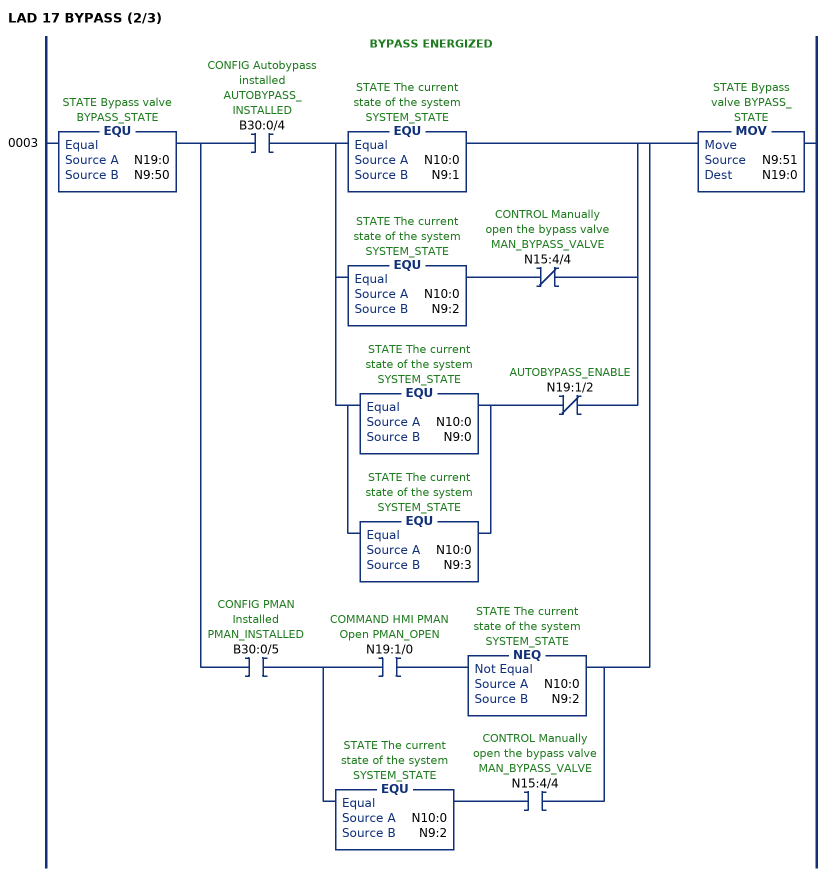
% Rung: 3 %
% TITLE: BYPASS ENERGIZED %
SOR EQU N19:0 N9:50 BST XIC B30:0/4 BST EQU N10:0 N9:1 NXB EQU N10:0 N9:2 XIO N15:4/4 NXB BST EQU N10:0 N9:0 NXB EQU N10:0 N9:3 BND XIO N19:1/2 BND NXB XIC B30:0/5 BST XIC N19:1/0 NEQ N10:0 N9:2 NXB EQU N10:0 N9:2 XIC N15:4/4 BND BND MOV N9:51 N19:0 EOR
%   N19:0  BYPASS_STATE  "STATE Bypass valve" %
%   N9:50  BYPASS_DEENERGIZED  "STATE Bypass Deenergized" %
%   B30:0/4  AUTOBYPASS_INSTALLED  "CONFIG Autobypass installed" %
%   N10:0  SYSTEM_STATE  "STATE The current state of the system" %
%   N9:1  SYSTEM_PROCESS  "STATE System Process" %
%   N9:2  SYSTEM_MANUAL  "STATE System Manual" %
%   N15:4/4  MAN_BYPASS_VALVE  "CONTROL Manually open the bypass valve" %
%   N9:0  SYSTEM_STANDBY  "STATE System Standby" %
%   N9:3  SYSTEM_ALARM  "STATE System Alarm" %
%   N19:1/2  AUTOBYPASS_ENABLE %
%   B30:0/5  PMAN_INSTALLED  "CONFIG PMAN Installed" %
%   N19:1/0  PMAN_OPEN  "COMMAND HMI PMAN Open" %
%   N9:51  BYPASS_ENERGIZED  "STATE Bypass Energized" %

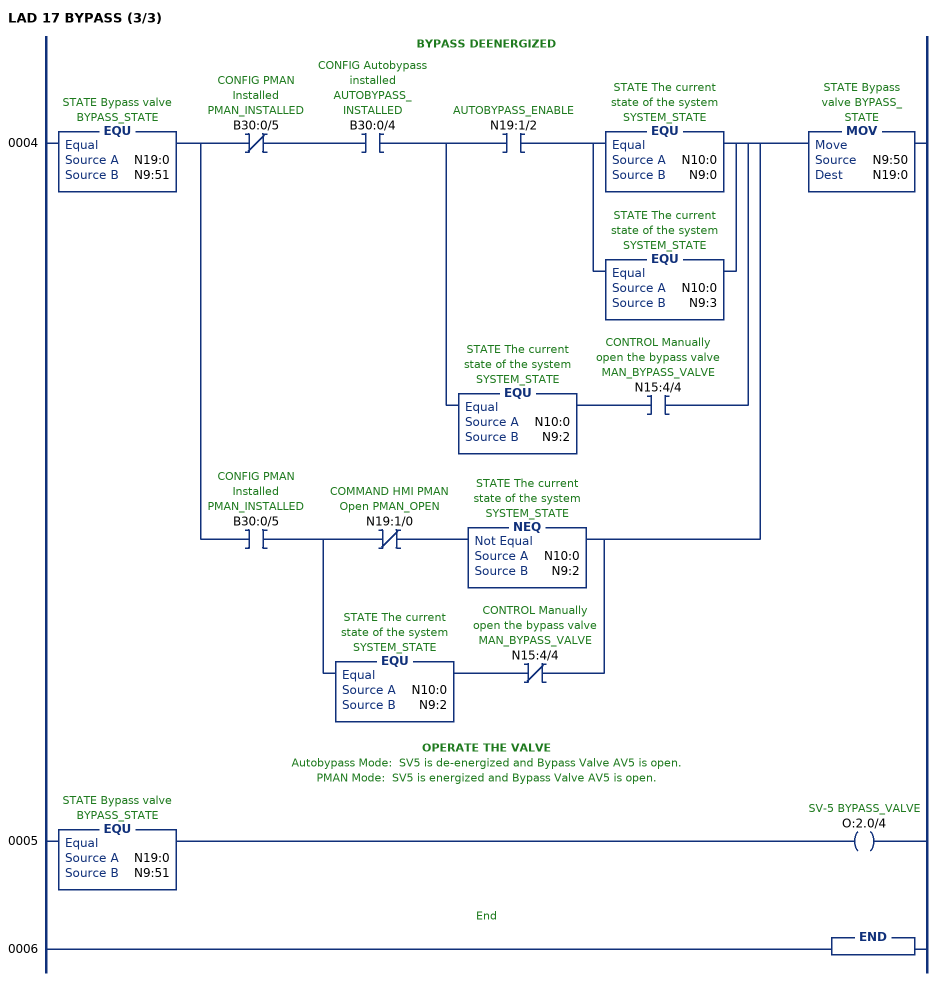
% Rung: 4 %
% TITLE: BYPASS DEENERGIZED %
SOR EQU N19:0 N9:51 BST XIO B30:0/5 XIC B30:0/4 BST XIC N19:1/2 BST EQU N10:0 N9:0 NXB EQU N10:0 N9:3 BND NXB EQU N10:0 N9:2 XIC N15:4/4 BND NXB XIC B30:0/5 BST XIO N19:1/0 NEQ N10:0 N9:2 NXB EQU N10:0 N9:2 XIO N15:4/4 BND BND MOV N9:50 N19:0 EOR
%   N19:0  BYPASS_STATE  "STATE Bypass valve" %
%   N9:51  BYPASS_ENERGIZED  "STATE Bypass Energized" %
%   B30:0/5  PMAN_INSTALLED  "CONFIG PMAN Installed" %
%   B30:0/4  AUTOBYPASS_INSTALLED  "CONFIG Autobypass installed" %
%   N19:1/2  AUTOBYPASS_ENABLE %
%   N10:0  SYSTEM_STATE  "STATE The current state of the system" %
%   N9:0  SYSTEM_STANDBY  "STATE System Standby" %
%   N9:3  SYSTEM_ALARM  "STATE System Alarm" %
%   N9:2  SYSTEM_MANUAL  "STATE System Manual" %
%   N15:4/4  MAN_BYPASS_VALVE  "CONTROL Manually open the bypass valve" %
%   N19:1/0  PMAN_OPEN  "COMMAND HMI PMAN Open" %
%   N9:50  BYPASS_DEENERGIZED  "STATE Bypass Deenergized" %
% Rung: 5 %
% TITLE: OPERATE THE VALVE %
% Autobypass Mode:  SV5 is de-energized and Bypass Valve AV5 is open.
% PMAN Mode:  SV5 is energized and Bypass Valve AV5 is open. %
SOR EQU N19:0 N9:51 OTE O:2.0/4 EOR
%   N19:0  BYPASS_STATE  "STATE Bypass valve" %
%   N9:51  BYPASS_ENERGIZED  "STATE Bypass Energized" %
%   O:2.0/4  BYPASS_VALVE  "SV-5" %
% Rung: 6 %
% End %
SOR END EOR

LADDER 18 "MIX PANEL"
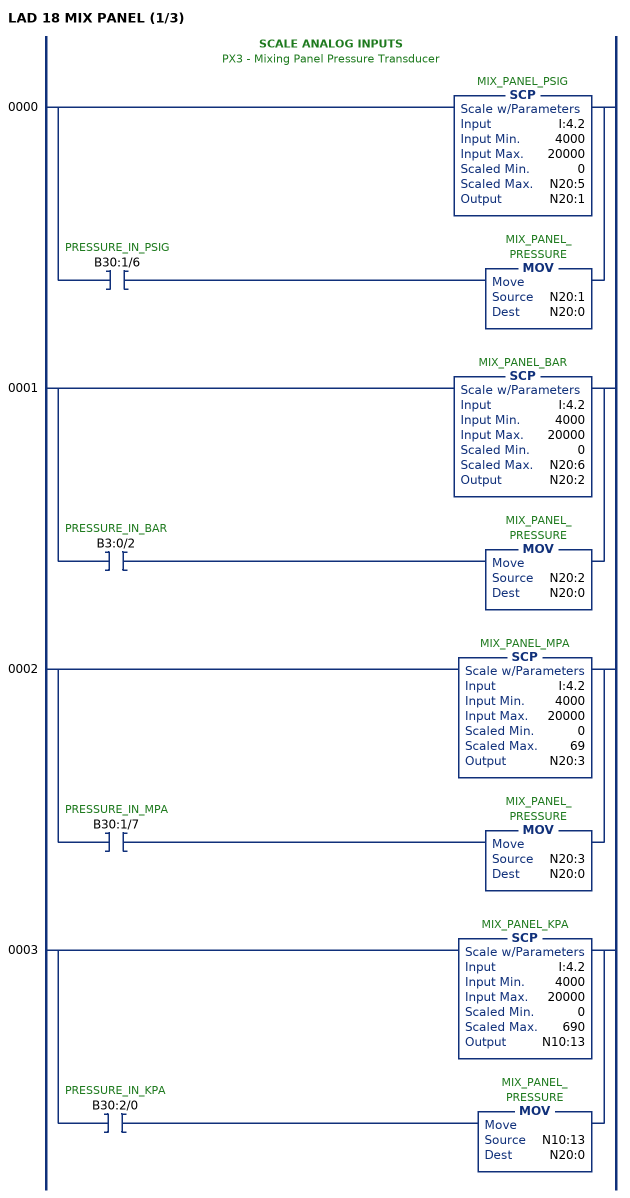
% Rung: 0 %
% TITLE: SCALE ANALOG INPUTS %
% PX3 - Mixing Panel Pressure Transducer %
SOR BST SCP I:4.2 4000 20000 0 N20:5 N20:1 NXB XIC B30:1/6 MOV N20:1 N20:0 BND EOR
%   I:4.2  MIX_PANEL_PX_READING  "PX-3" %
%   N20:5  PX3_SCALING %
%   N20:1  MIX_PANEL_PSIG %
%   B30:1/6  PRESSURE_IN_PSIG %
%   N20:0  MIX_PANEL_PRESSURE %
% Rung: 1 %
SOR BST SCP I:4.2 4000 20000 0 N20:6 N20:2 NXB XIC B3:0/2 MOV N20:2 N20:0 BND EOR
%   I:4.2  MIX_PANEL_PX_READING  "PX-3" %
%   N20:6  PX3_SCALING_BAR %
%   N20:2  MIX_PANEL_BAR %
%   B3:0/2  PRESSURE_IN_BAR %
%   N20:0  MIX_PANEL_PRESSURE %
% Rung: 2 %
SOR BST SCP I:4.2 4000 20000 0 69 N20:3 NXB XIC B30:1/7 MOV N20:3 N20:0 BND EOR
%   I:4.2  MIX_PANEL_PX_READING  "PX-3" %
%   N20:3  MIX_PANEL_MPA %
%   B30:1/7  PRESSURE_IN_MPA %
%   N20:0  MIX_PANEL_PRESSURE %
% Rung: 3 %
SOR BST SCP I:4.2 4000 20000 0 690 N10:13 NXB XIC B30:2/0 MOV N10:13 N20:0 BND EOR
%   I:4.2  MIX_PANEL_PX_READING  "PX-3" %
%   N10:13  MIX_PANEL_KPA %
%   B30:2/0  PRESSURE_IN_KPA %
%   N20:0  MIX_PANEL_PRESSURE %

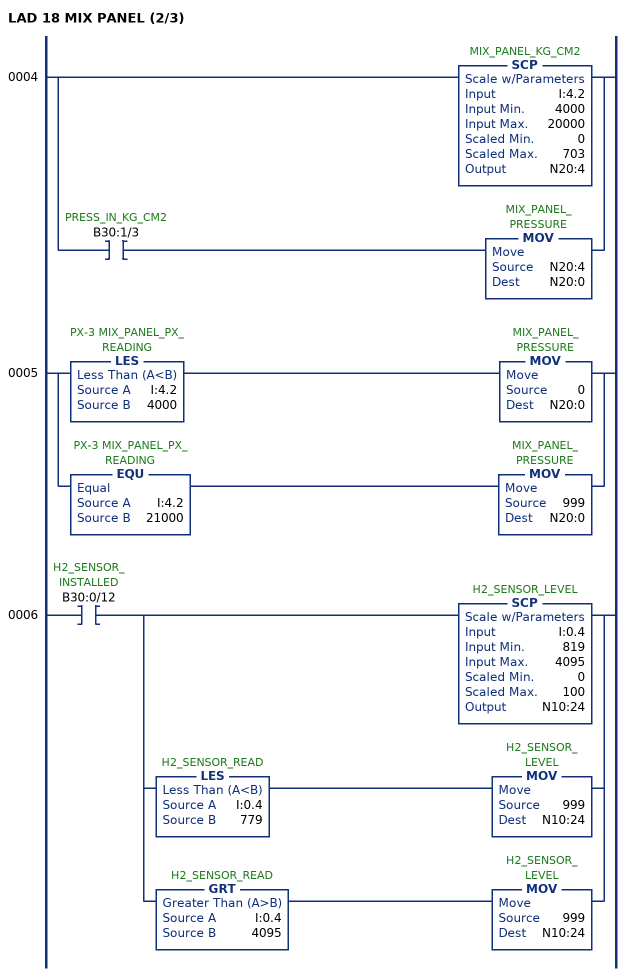
% Rung: 4 %
SOR BST SCP I:4.2 4000 20000 0 703 N20:4 NXB XIC B30:1/3 MOV N20:4 N20:0 BND EOR
%   I:4.2  MIX_PANEL_PX_READING  "PX-3" %
%   N20:4  MIX_PANEL_KG_CM2 %
%   B30:1/3  PRESS_IN_KG_CM2 %
%   N20:0  MIX_PANEL_PRESSURE %
% Rung: 5 %
SOR BST LES I:4.2 4000 MOV 0 N20:0 NXB EQU I:4.2 21000 MOV 999 N20:0 BND EOR
%   I:4.2  MIX_PANEL_PX_READING  "PX-3" %
%   N20:0  MIX_PANEL_PRESSURE %
% Rung: 6 %
SOR XIC B30:0/12 BST SCP I:0.4 819 4095 0 100 N10:24 NXB LES I:0.4 779 MOV 999 N10:24 NXB GRT I:0.4 4095 MOV 999 N10:24 BND EOR
%   B30:0/12  H2_SENSOR_INSTALLED %
%   I:0.4  H2_SENSOR_READ %
%   N10:24  H2_SENSOR_LEVEL %

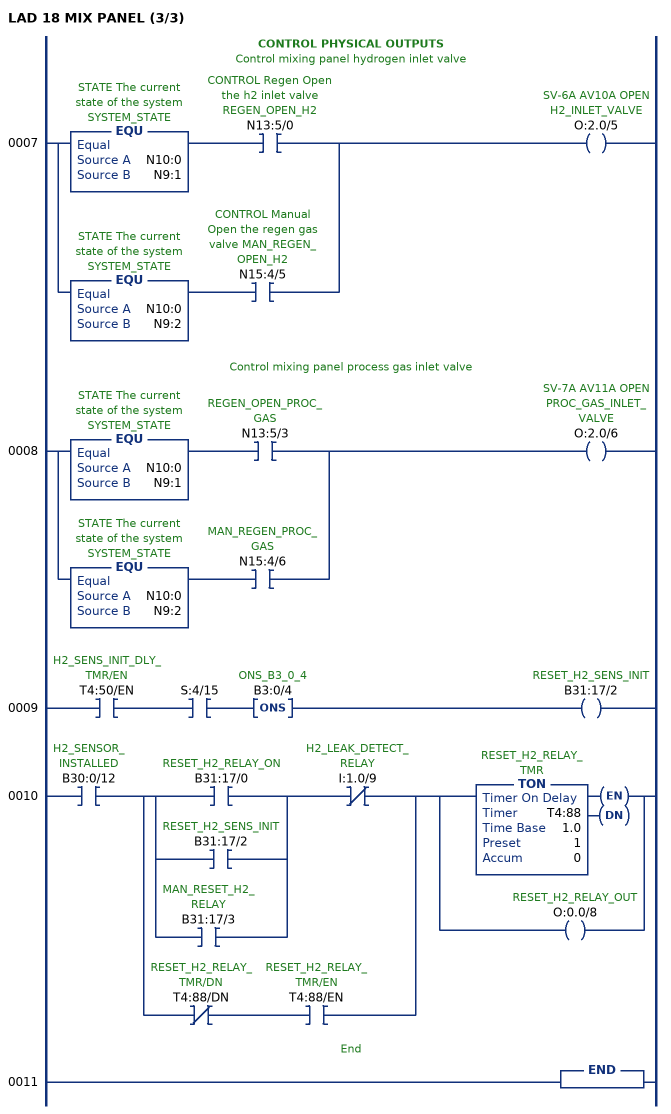
% Rung: 7 %
% TITLE: CONTROL PHYSICAL OUTPUTS %
% Control mixing panel hydrogen inlet valve %
SOR BST EQU N10:0 N9:1 XIC N13:5/0 NXB EQU N10:0 N9:2 XIC N15:4/5 BND OTE O:2.0/5 EOR
%   N10:0  SYSTEM_STATE  "STATE The current state of the system" %
%   N9:1  SYSTEM_PROCESS  "STATE System Process" %
%   N13:5/0  REGEN_OPEN_H2  "CONTROL Regen Open the h2 inlet valve" %
%   N9:2  SYSTEM_MANUAL  "STATE System Manual" %
%   N15:4/5  MAN_REGEN_OPEN_H2  "CONTROL Manual Open the regen gas valve" %
%   O:2.0/5  H2_INLET_VALVE  "SV-6A AV10A OPEN" %
% Rung: 8 %
% Control mixing panel process gas inlet valve %
SOR BST EQU N10:0 N9:1 XIC N13:5/3 NXB EQU N10:0 N9:2 XIC N15:4/6 BND OTE O:2.0/6 EOR
%   N10:0  SYSTEM_STATE  "STATE The current state of the system" %
%   N9:1  SYSTEM_PROCESS  "STATE System Process" %
%   N13:5/3  REGEN_OPEN_PROC_GAS %
%   N9:2  SYSTEM_MANUAL  "STATE System Manual" %
%   N15:4/6  MAN_REGEN_PROC_GAS %
%   O:2.0/6  PROC_GAS_INLET_VALVE  "SV-7A AV11A OPEN" %
% Rung: 9 %
SOR XIC T4:50/EN XIC S:4/15 ONS B3:0/4 OTE B31:17/2 EOR
%   T4:50  H2_SENS_INIT_DLY_TMR %
%   B3:0/4  ONS_B3_0_4 %
%   B31:17/2  RESET_H2_SENS_INIT %
% Rung: 10 %
SOR XIC B30:0/12 BST BST XIC B31:17/0 NXB XIC B31:17/2 NXB XIC B31:17/3 BND XIO I:1.0/9 NXB XIO T4:88/DN XIC T4:88/EN BND BST TON T4:88 1.0 1 0 NXB OTE O:0.0/8 BND EOR
%   B30:0/12  H2_SENSOR_INSTALLED %
%   B31:17/0  RESET_H2_RELAY_ON %
%   B31:17/2  RESET_H2_SENS_INIT %
%   B31:17/3  MAN_RESET_H2_RELAY %
%   I:1.0/9  H2_LEAK_DETECT_RELAY %
%   T4:88  RESET_H2_RELAY_TMR %
%   O:0.0/8  RESET_H2_RELAY_OUT %
% Rung: 11 %
% End %
SOR END EOR

LADDER 20 "ADS_A"    % Controls the Adsorber A %
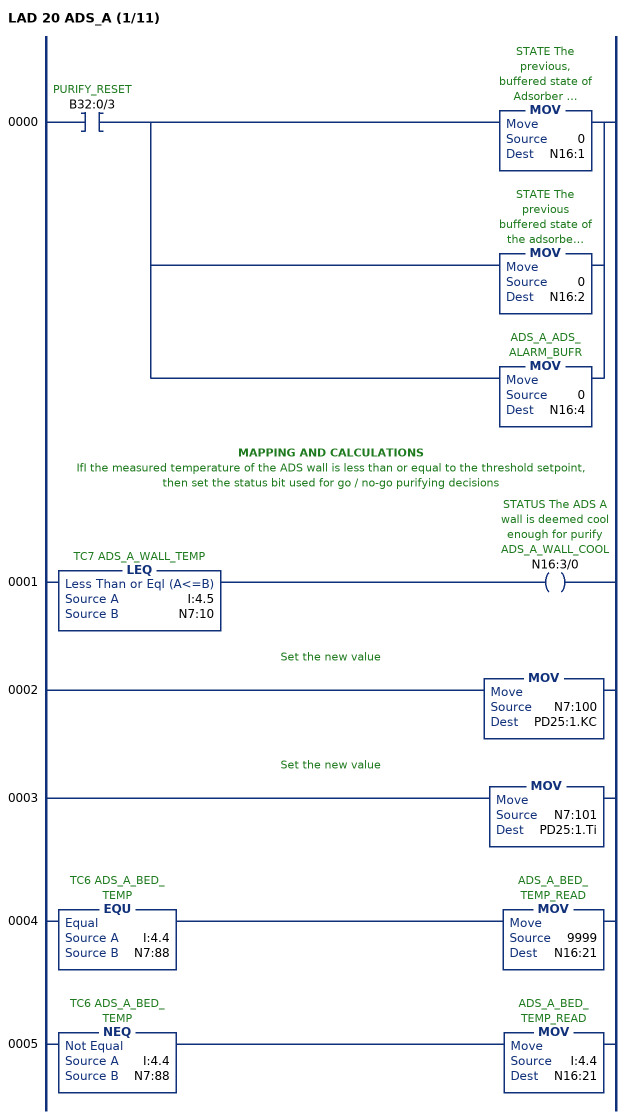
% Rung: 0 %
SOR XIC B32:0/3 BST MOV 0 N16:1 NXB MOV 0 N16:2 NXB MOV 0 N16:4 BND EOR
%   B32:0/3  PURIFY_RESET %
%   N16:1  ADS_A_STANDBY_BUFFER  "STATE The previous, buffered state of Adsorber A" %
%   N16:2  ADS_A_SYS_ALARM_BUFR  "STATE The previous buffered state of the adsorber when the alarm occured" %
%   N16:4  ADS_A_ADS_ALARM_BUFR %
% Rung: 1 %
% TITLE: MAPPING AND CALCULATIONS %
% IfI the measured temperature of the ADS wall is less than or equal to the threshold setpoint, then set the status bit used for go / no-go purifying decisions %
SOR LEQ I:4.5 N7:10 OTE N16:3/0 EOR
%   I:4.5  ADS_A_WALL_TEMP  "TC7" %
%   N7:10  ADS_WALL_TEMP_COOL  "CONFIG The temp at which the adsorber wall is deemed to be cool enough to purify" %
%   N16:3/0  ADS_A_WALL_COOL  "STATUS The ADS A wall is deemed cool enough for purify" %
% Rung: 2 %
% Set the new value %
SOR MOV N7:100 PD25:1.KC EOR
%   N7:100  BLANKET_P  "CONFIG Blanket Proportional Gain New" %
% Rung: 3 %
% Set the new value %
SOR MOV N7:101 PD25:1.Ti EOR
%   N7:101  BLANKET_I  "CONFIG Blanket Integral Gain New" %
% Rung: 4 %
SOR EQU I:4.4 N7:88 MOV 9999 N16:21 EOR
%   I:4.4  ADS_A_BED_TEMP  "TC6" %
%   N7:88  TC_OPEN_SP  "CONFIG The value read by an open TC input" %
%   N16:21  ADS_A_BED_TEMP_READ %
% Rung: 5 %
SOR NEQ I:4.4 N7:88 MOV I:4.4 N16:21 EOR
%   I:4.4  ADS_A_BED_TEMP  "TC6" %
%   N7:88  TC_OPEN_SP  "CONFIG The value read by an open TC input" %
%   N16:21  ADS_A_BED_TEMP_READ %

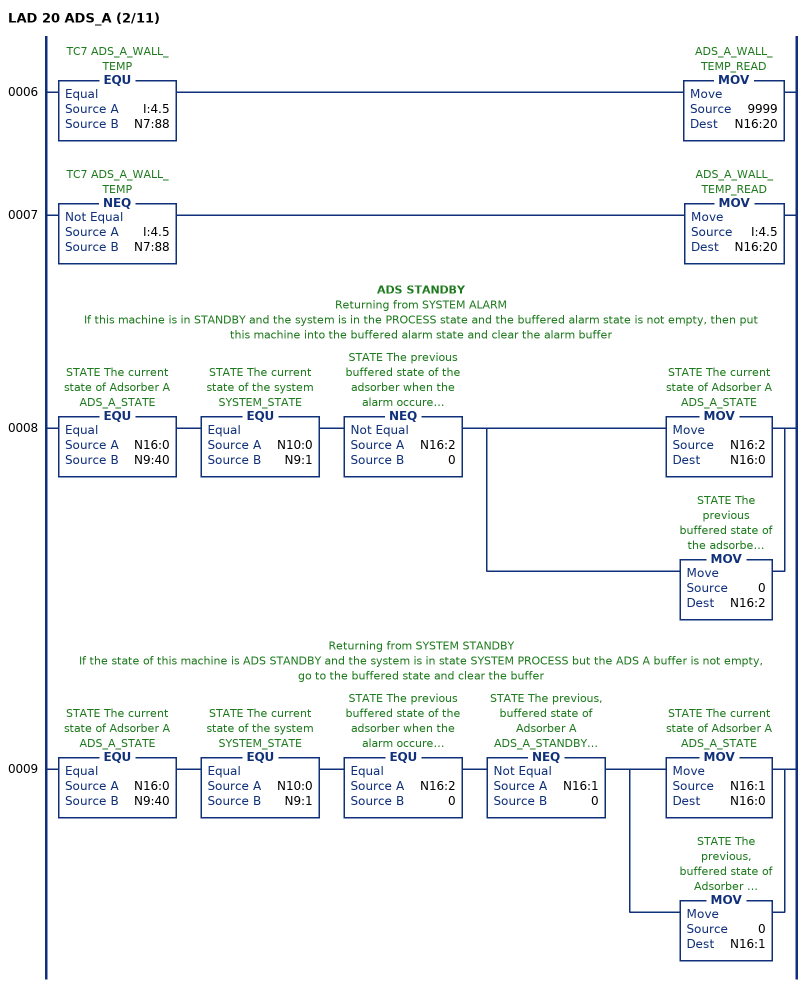
% Rung: 6 %
SOR EQU I:4.5 N7:88 MOV 9999 N16:20 EOR
%   I:4.5  ADS_A_WALL_TEMP  "TC7" %
%   N7:88  TC_OPEN_SP  "CONFIG The value read by an open TC input" %
%   N16:20  ADS_A_WALL_TEMP_READ %
% Rung: 7 %
SOR NEQ I:4.5 N7:88 MOV I:4.5 N16:20 EOR
%   I:4.5  ADS_A_WALL_TEMP  "TC7" %
%   N7:88  TC_OPEN_SP  "CONFIG The value read by an open TC input" %
%   N16:20  ADS_A_WALL_TEMP_READ %
% Rung: 8 %
% TITLE: ADS STANDBY %
% Returning from SYSTEM ALARM
% If this machine is in STANDBY and the system is in the PROCESS state and the buffered alarm state is not empty, then put this machine into the buffered alarm state and clear the alarm buffer %
SOR EQU N16:0 N9:40 EQU N10:0 N9:1 NEQ N16:2 0 BST MOV N16:2 N16:0 NXB MOV 0 N16:2 BND EOR
%   N16:0  ADS_A_STATE  "STATE The current state of Adsorber A" %
%   N9:40  ADS_STANDBY  "STATE ADS Standby" %
%   N10:0  SYSTEM_STATE  "STATE The current state of the system" %
%   N9:1  SYSTEM_PROCESS  "STATE System Process" %
%   N16:2  ADS_A_SYS_ALARM_BUFR  "STATE The previous buffered state of the adsorber when the alarm occured" %
% Rung: 9 %
% Returning from SYSTEM STANDBY
% If the state of this machine is ADS STANDBY and the system is in state SYSTEM PROCESS but the ADS A buffer is not empty, go to the buffered state and clear the buffer %
SOR EQU N16:0 N9:40 EQU N10:0 N9:1 EQU N16:2 0 NEQ N16:1 0 BST MOV N16:1 N16:0 NXB MOV 0 N16:1 BND EOR
%   N16:0  ADS_A_STATE  "STATE The current state of Adsorber A" %
%   N9:40  ADS_STANDBY  "STATE ADS Standby" %
%   N10:0  SYSTEM_STATE  "STATE The current state of the system" %
%   N9:1  SYSTEM_PROCESS  "STATE System Process" %
%   N16:2  ADS_A_SYS_ALARM_BUFR  "STATE The previous buffered state of the adsorber when the alarm occured" %
%   N16:1  ADS_A_STANDBY_BUFFER  "STATE The previous, buffered state of Adsorber A" %

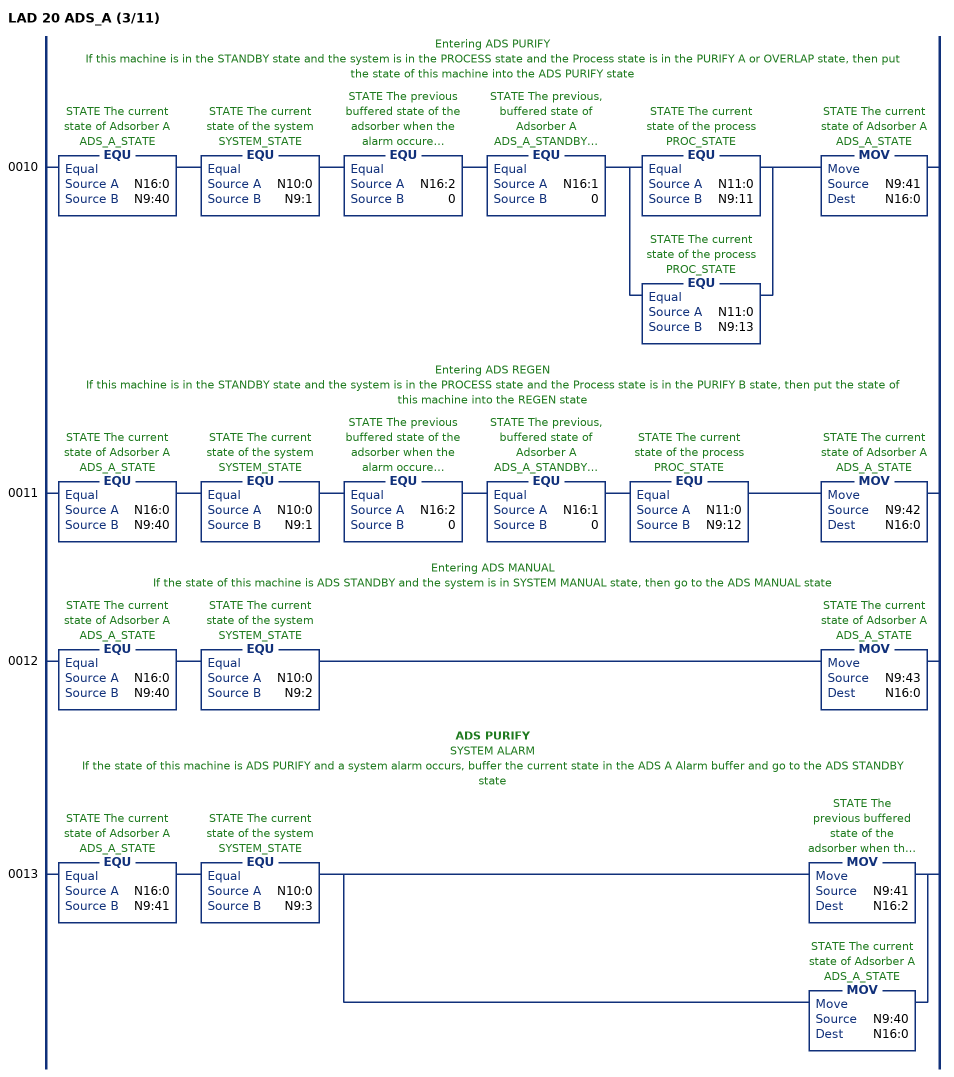
% Rung: 10 %
% Entering ADS PURIFY
% If this machine is in the STANDBY state and the system is in the PROCESS state and the Process state is in the PURIFY A or OVERLAP state, then put the state of this machine into the ADS PURIFY state %
SOR EQU N16:0 N9:40 EQU N10:0 N9:1 EQU N16:2 0 EQU N16:1 0 BST EQU N11:0 N9:11 NXB EQU N11:0 N9:13 BND MOV N9:41 N16:0 EOR
%   N16:0  ADS_A_STATE  "STATE The current state of Adsorber A" %
%   N9:40  ADS_STANDBY  "STATE ADS Standby" %
%   N10:0  SYSTEM_STATE  "STATE The current state of the system" %
%   N9:1  SYSTEM_PROCESS  "STATE System Process" %
%   N16:2  ADS_A_SYS_ALARM_BUFR  "STATE The previous buffered state of the adsorber when the alarm occured" %
%   N16:1  ADS_A_STANDBY_BUFFER  "STATE The previous, buffered state of Adsorber A" %
%   N11:0  PROC_STATE  "STATE The current state of the process" %
%   N9:11  PROC_PURIFY_A  "STATE Process Purify A" %
%   N9:13  PROC_OVERLAP  "STATE Process Purify Overlap" %
%   N9:41  ADS_PURIFY  "STATE ADS Purify" %
% Rung: 11 %
% Entering ADS REGEN
% If this machine is in the STANDBY state and the system is in the PROCESS state and the Process state is in the PURIFY B state, then put the state of this machine into the REGEN state %
SOR EQU N16:0 N9:40 EQU N10:0 N9:1 EQU N16:2 0 EQU N16:1 0 EQU N11:0 N9:12 MOV N9:42 N16:0 EOR
%   N16:0  ADS_A_STATE  "STATE The current state of Adsorber A" %
%   N9:40  ADS_STANDBY  "STATE ADS Standby" %
%   N10:0  SYSTEM_STATE  "STATE The current state of the system" %
%   N9:1  SYSTEM_PROCESS  "STATE System Process" %
%   N16:2  ADS_A_SYS_ALARM_BUFR  "STATE The previous buffered state of the adsorber when the alarm occured" %
%   N16:1  ADS_A_STANDBY_BUFFER  "STATE The previous, buffered state of Adsorber A" %
%   N11:0  PROC_STATE  "STATE The current state of the process" %
%   N9:12  PROC_PURIFY_B  "STATE Process Purify B" %
%   N9:42  ADS_REGEN  "STATE ADS Regen" %
% Rung: 12 %
% Entering ADS MANUAL
% If the state of this machine is ADS STANDBY and the system is in SYSTEM MANUAL state, then go to the ADS MANUAL state %
SOR EQU N16:0 N9:40 EQU N10:0 N9:2 MOV N9:43 N16:0 EOR
%   N16:0  ADS_A_STATE  "STATE The current state of Adsorber A" %
%   N9:40  ADS_STANDBY  "STATE ADS Standby" %
%   N10:0  SYSTEM_STATE  "STATE The current state of the system" %
%   N9:2  SYSTEM_MANUAL  "STATE System Manual" %
%   N9:43  ADS_MANUAL  "STATE ADS Manual" %
% Rung: 13 %
% TITLE: ADS PURIFY %
% SYSTEM ALARM
% If the state of this machine is ADS PURIFY and a system alarm occurs, buffer the current state in the ADS A Alarm buffer and go to the ADS STANDBY state %
SOR EQU N16:0 N9:41 EQU N10:0 N9:3 BST MOV N9:41 N16:2 NXB MOV N9:40 N16:0 BND EOR
%   N16:0  ADS_A_STATE  "STATE The current state of Adsorber A" %
%   N9:41  ADS_PURIFY  "STATE ADS Purify" %
%   N10:0  SYSTEM_STATE  "STATE The current state of the system" %
%   N9:3  SYSTEM_ALARM  "STATE System Alarm" %
%   N16:2  ADS_A_SYS_ALARM_BUFR  "STATE The previous buffered state of the adsorber when the alarm occured" %
%   N9:40  ADS_STANDBY  "STATE ADS Standby" %

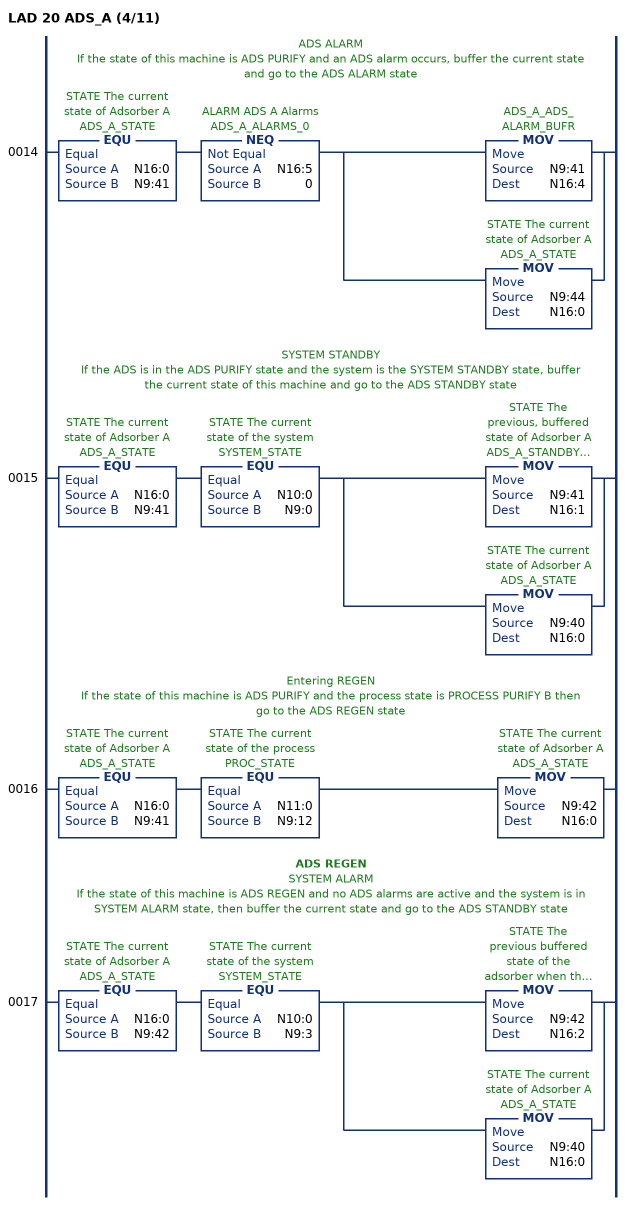
% Rung: 14 %
% ADS ALARM
% If the state of this machine is ADS PURIFY and an ADS alarm occurs, buffer the current state and go to the ADS ALARM state %
SOR EQU N16:0 N9:41 NEQ N16:5 0 BST MOV N9:41 N16:4 NXB MOV N9:44 N16:0 BND EOR
%   N16:0  ADS_A_STATE  "STATE The current state of Adsorber A" %
%   N9:41  ADS_PURIFY  "STATE ADS Purify" %
%   N16:5  ADS_A_ALARMS_0  "ALARM ADS A Alarms" %
%   N16:4  ADS_A_ADS_ALARM_BUFR %
%   N9:44  ADS_ALARM  "STATE ADS Alarm" %
% Rung: 15 %
% SYSTEM STANDBY
% If the ADS is in the ADS PURIFY state and the system is the SYSTEM STANDBY state, buffer the current state of this machine and go to the ADS STANDBY state %
SOR EQU N16:0 N9:41 EQU N10:0 N9:0 BST MOV N9:41 N16:1 NXB MOV N9:40 N16:0 BND EOR
%   N16:0  ADS_A_STATE  "STATE The current state of Adsorber A" %
%   N9:41  ADS_PURIFY  "STATE ADS Purify" %
%   N10:0  SYSTEM_STATE  "STATE The current state of the system" %
%   N9:0  SYSTEM_STANDBY  "STATE System Standby" %
%   N16:1  ADS_A_STANDBY_BUFFER  "STATE The previous, buffered state of Adsorber A" %
%   N9:40  ADS_STANDBY  "STATE ADS Standby" %
% Rung: 16 %
% Entering REGEN
% If the state of this machine is ADS PURIFY and the process state is PROCESS PURIFY B then go to the ADS REGEN state %
SOR EQU N16:0 N9:41 EQU N11:0 N9:12 MOV N9:42 N16:0 EOR
%   N16:0  ADS_A_STATE  "STATE The current state of Adsorber A" %
%   N9:41  ADS_PURIFY  "STATE ADS Purify" %
%   N11:0  PROC_STATE  "STATE The current state of the process" %
%   N9:12  PROC_PURIFY_B  "STATE Process Purify B" %
%   N9:42  ADS_REGEN  "STATE ADS Regen" %
% Rung: 17 %
% TITLE: ADS REGEN %
% SYSTEM ALARM
% If the state of this machine is ADS REGEN and no ADS alarms are active and the system is in SYSTEM ALARM state, then buffer the current state and go to the ADS STANDBY state %
SOR EQU N16:0 N9:42 EQU N10:0 N9:3 BST MOV N9:42 N16:2 NXB MOV N9:40 N16:0 BND EOR
%   N16:0  ADS_A_STATE  "STATE The current state of Adsorber A" %
%   N9:42  ADS_REGEN  "STATE ADS Regen" %
%   N10:0  SYSTEM_STATE  "STATE The current state of the system" %
%   N9:3  SYSTEM_ALARM  "STATE System Alarm" %
%   N16:2  ADS_A_SYS_ALARM_BUFR  "STATE The previous buffered state of the adsorber when the alarm occured" %
%   N9:40  ADS_STANDBY  "STATE ADS Standby" %

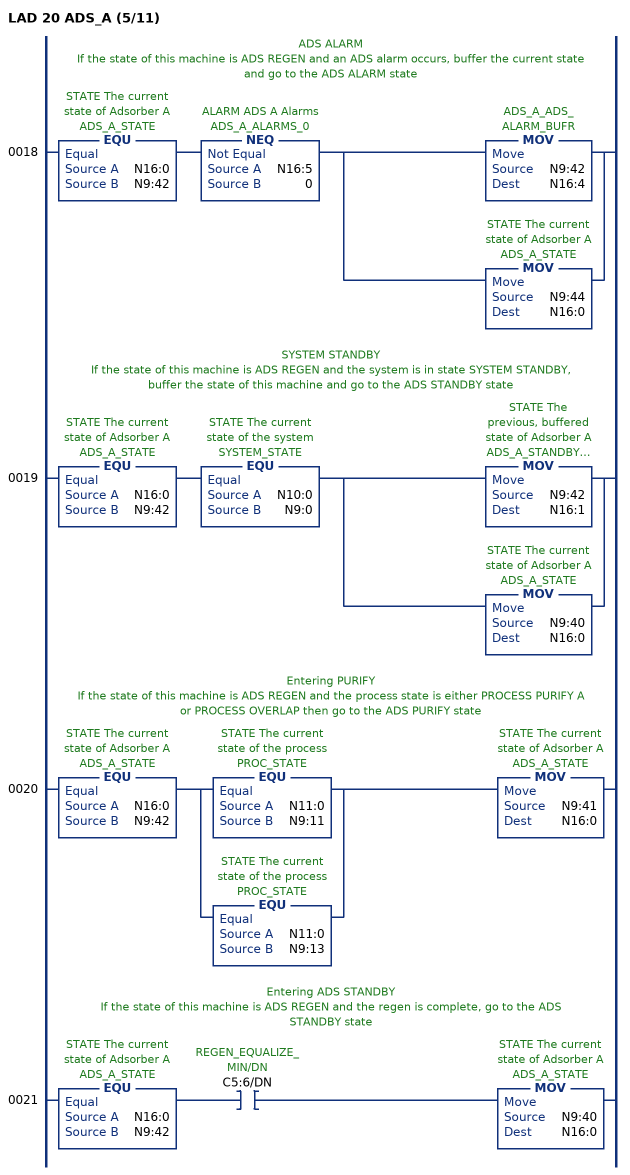
% Rung: 18 %
% ADS ALARM
% If the state of this machine is ADS REGEN and an ADS alarm occurs, buffer the current state and go to the ADS ALARM state %
SOR EQU N16:0 N9:42 NEQ N16:5 0 BST MOV N9:42 N16:4 NXB MOV N9:44 N16:0 BND EOR
%   N16:0  ADS_A_STATE  "STATE The current state of Adsorber A" %
%   N9:42  ADS_REGEN  "STATE ADS Regen" %
%   N16:5  ADS_A_ALARMS_0  "ALARM ADS A Alarms" %
%   N16:4  ADS_A_ADS_ALARM_BUFR %
%   N9:44  ADS_ALARM  "STATE ADS Alarm" %
% Rung: 19 %
% SYSTEM STANDBY
% If the state of this machine is ADS REGEN and the system is in state SYSTEM STANDBY, buffer the state of this machine and go to the ADS STANDBY state %
SOR EQU N16:0 N9:42 EQU N10:0 N9:0 BST MOV N9:42 N16:1 NXB MOV N9:40 N16:0 BND EOR
%   N16:0  ADS_A_STATE  "STATE The current state of Adsorber A" %
%   N9:42  ADS_REGEN  "STATE ADS Regen" %
%   N10:0  SYSTEM_STATE  "STATE The current state of the system" %
%   N9:0  SYSTEM_STANDBY  "STATE System Standby" %
%   N16:1  ADS_A_STANDBY_BUFFER  "STATE The previous, buffered state of Adsorber A" %
%   N9:40  ADS_STANDBY  "STATE ADS Standby" %
% Rung: 20 %
% Entering PURIFY
% If the state of this machine is ADS REGEN and the process state is either PROCESS PURIFY A or PROCESS OVERLAP then go to the ADS PURIFY state %
SOR EQU N16:0 N9:42 BST EQU N11:0 N9:11 NXB EQU N11:0 N9:13 BND MOV N9:41 N16:0 EOR
%   N16:0  ADS_A_STATE  "STATE The current state of Adsorber A" %
%   N9:42  ADS_REGEN  "STATE ADS Regen" %
%   N11:0  PROC_STATE  "STATE The current state of the process" %
%   N9:11  PROC_PURIFY_A  "STATE Process Purify A" %
%   N9:13  PROC_OVERLAP  "STATE Process Purify Overlap" %
%   N9:41  ADS_PURIFY  "STATE ADS Purify" %
% Rung: 21 %
% Entering ADS STANDBY
% If the state of this machine is ADS REGEN and the regen is complete, go to the ADS STANDBY state %
SOR EQU N16:0 N9:42 XIC C5:6/DN MOV N9:40 N16:0 EOR
%   N16:0  ADS_A_STATE  "STATE The current state of Adsorber A" %
%   N9:42  ADS_REGEN  "STATE ADS Regen" %
%   C5:6  REGEN_EQUALIZE_MIN %
%   N9:40  ADS_STANDBY  "STATE ADS Standby" %

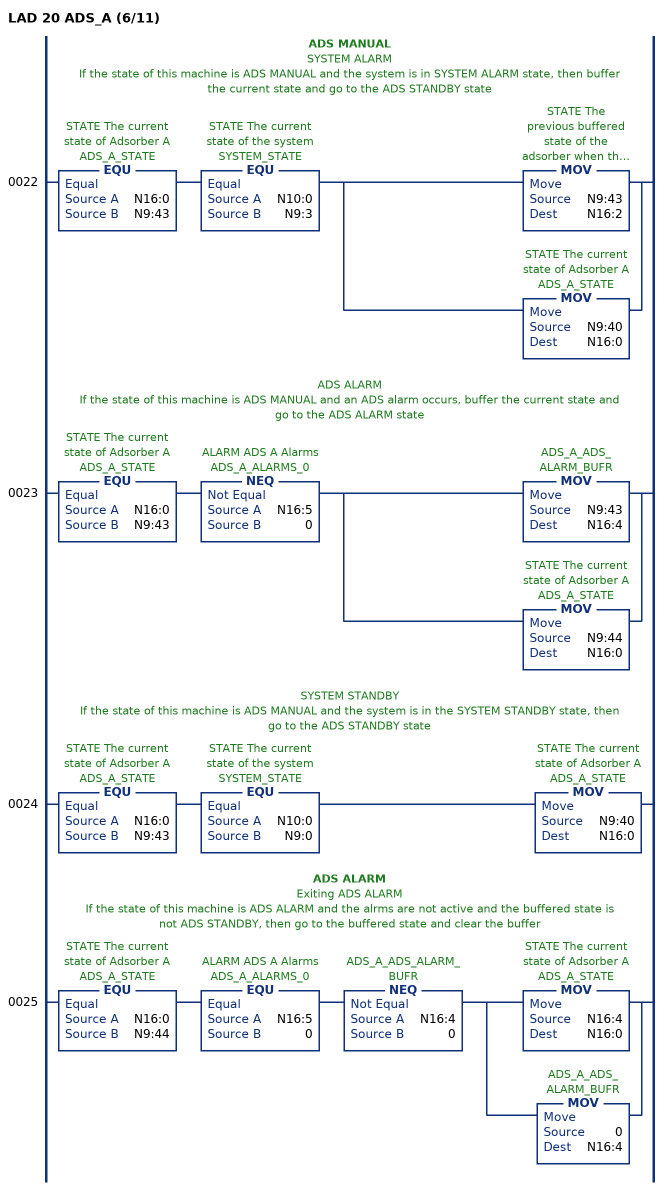
% Rung: 22 %
% TITLE: ADS MANUAL %
% SYSTEM ALARM
% If the state of this machine is ADS MANUAL and the system is in SYSTEM ALARM state, then buffer the current state and go to the ADS STANDBY state %
SOR EQU N16:0 N9:43 EQU N10:0 N9:3 BST MOV N9:43 N16:2 NXB MOV N9:40 N16:0 BND EOR
%   N16:0  ADS_A_STATE  "STATE The current state of Adsorber A" %
%   N9:43  ADS_MANUAL  "STATE ADS Manual" %
%   N10:0  SYSTEM_STATE  "STATE The current state of the system" %
%   N9:3  SYSTEM_ALARM  "STATE System Alarm" %
%   N16:2  ADS_A_SYS_ALARM_BUFR  "STATE The previous buffered state of the adsorber when the alarm occured" %
%   N9:40  ADS_STANDBY  "STATE ADS Standby" %
% Rung: 23 %
% ADS ALARM
% If the state of this machine is ADS MANUAL and an ADS alarm occurs, buffer the current state and go to the ADS ALARM state %
SOR EQU N16:0 N9:43 NEQ N16:5 0 BST MOV N9:43 N16:4 NXB MOV N9:44 N16:0 BND EOR
%   N16:0  ADS_A_STATE  "STATE The current state of Adsorber A" %
%   N9:43  ADS_MANUAL  "STATE ADS Manual" %
%   N16:5  ADS_A_ALARMS_0  "ALARM ADS A Alarms" %
%   N16:4  ADS_A_ADS_ALARM_BUFR %
%   N9:44  ADS_ALARM  "STATE ADS Alarm" %
% Rung: 24 %
% SYSTEM STANDBY
% If the state of this machine is ADS MANUAL and the system is in the SYSTEM STANDBY state, then go to the ADS STANDBY state %
SOR EQU N16:0 N9:43 EQU N10:0 N9:0 MOV N9:40 N16:0 EOR
%   N16:0  ADS_A_STATE  "STATE The current state of Adsorber A" %
%   N9:43  ADS_MANUAL  "STATE ADS Manual" %
%   N10:0  SYSTEM_STATE  "STATE The current state of the system" %
%   N9:0  SYSTEM_STANDBY  "STATE System Standby" %
%   N9:40  ADS_STANDBY  "STATE ADS Standby" %
% Rung: 25 %
% TITLE: ADS ALARM %
% Exiting ADS ALARM
% If the state of this machine is ADS ALARM and the alrms are not active and the buffered state is not ADS STANDBY, then go to the buffered state and clear the buffer %
SOR EQU N16:0 N9:44 EQU N16:5 0 NEQ N16:4 0 BST MOV N16:4 N16:0 NXB MOV 0 N16:4 BND EOR
%   N16:0  ADS_A_STATE  "STATE The current state of Adsorber A" %
%   N9:44  ADS_ALARM  "STATE ADS Alarm" %
%   N16:5  ADS_A_ALARMS_0  "ALARM ADS A Alarms" %
%   N16:4  ADS_A_ADS_ALARM_BUFR %

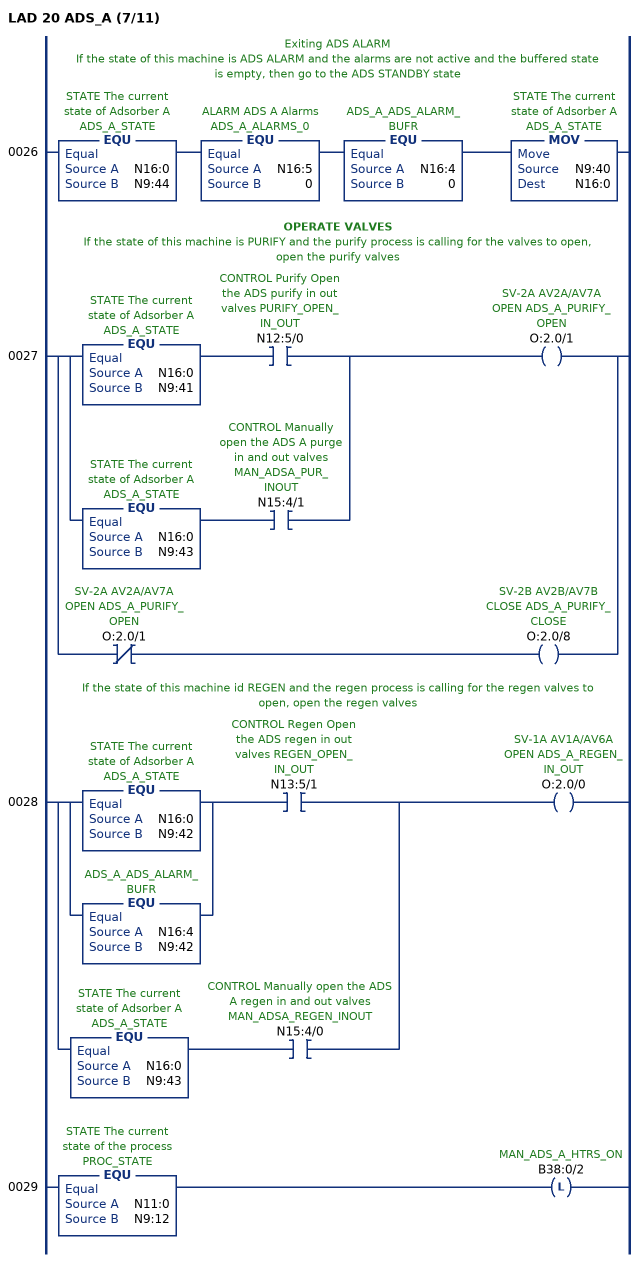
% Rung: 26 %
% Exiting ADS ALARM
% If the state of this machine is ADS ALARM and the alarms are not active and the buffered state is empty, then go to the ADS STANDBY state %
SOR EQU N16:0 N9:44 EQU N16:5 0 EQU N16:4 0 MOV N9:40 N16:0 EOR
%   N16:0  ADS_A_STATE  "STATE The current state of Adsorber A" %
%   N9:44  ADS_ALARM  "STATE ADS Alarm" %
%   N16:5  ADS_A_ALARMS_0  "ALARM ADS A Alarms" %
%   N16:4  ADS_A_ADS_ALARM_BUFR %
%   N9:40  ADS_STANDBY  "STATE ADS Standby" %
% Rung: 27 %
% TITLE: OPERATE VALVES %
% If the state of this machine is PURIFY and the purify process is calling for the valves to open, open the purify valves %
SOR BST BST EQU N16:0 N9:41 XIC N12:5/0 NXB EQU N16:0 N9:43 XIC N15:4/1 BND OTE O:2.0/1 NXB XIO O:2.0/1 OTE O:2.0/8 BND EOR
%   N16:0  ADS_A_STATE  "STATE The current state of Adsorber A" %
%   N9:41  ADS_PURIFY  "STATE ADS Purify" %
%   N12:5/0  PURIFY_OPEN_IN_OUT  "CONTROL Purify Open the ADS purify in out valves" %
%   N9:43  ADS_MANUAL  "STATE ADS Manual" %
%   N15:4/1  MAN_ADSA_PUR_INOUT  "CONTROL Manually open the ADS A purge in and out valves" %
%   O:2.0/1  ADS_A_PURIFY_OPEN  "SV-2A AV2A/AV7A OPEN" %
%   O:2.0/8  ADS_A_PURIFY_CLOSE  "SV-2B AV2B/AV7B CLOSE" %
% Rung: 28 %
% If the state of this machine id REGEN and the regen process is calling for the regen valves to open, open the regen valves %
SOR BST BST EQU N16:0 N9:42 NXB EQU N16:4 N9:42 BND XIC N13:5/1 NXB EQU N16:0 N9:43 XIC N15:4/0 BND OTE O:2.0/0 EOR
%   N16:0  ADS_A_STATE  "STATE The current state of Adsorber A" %
%   N9:42  ADS_REGEN  "STATE ADS Regen" %
%   N16:4  ADS_A_ADS_ALARM_BUFR %
%   N13:5/1  REGEN_OPEN_IN_OUT  "CONTROL Regen Open the ADS regen in out valves" %
%   N9:43  ADS_MANUAL  "STATE ADS Manual" %
%   N15:4/0  MAN_ADSA_REGEN_INOUT  "CONTROL Manually open the ADS A regen in and out valves" %
%   O:2.0/0  ADS_A_REGEN_IN_OUT  "SV-1A AV1A/AV6A OPEN" %
% Rung: 29 %
SOR EQU N11:0 N9:12 OTL B38:0/2 EOR
%   N11:0  PROC_STATE  "STATE The current state of the process" %
%   N9:12  PROC_PURIFY_B  "STATE Process Purify B" %
%   B38:0/2  MAN_ADS_A_HTRS_ON %

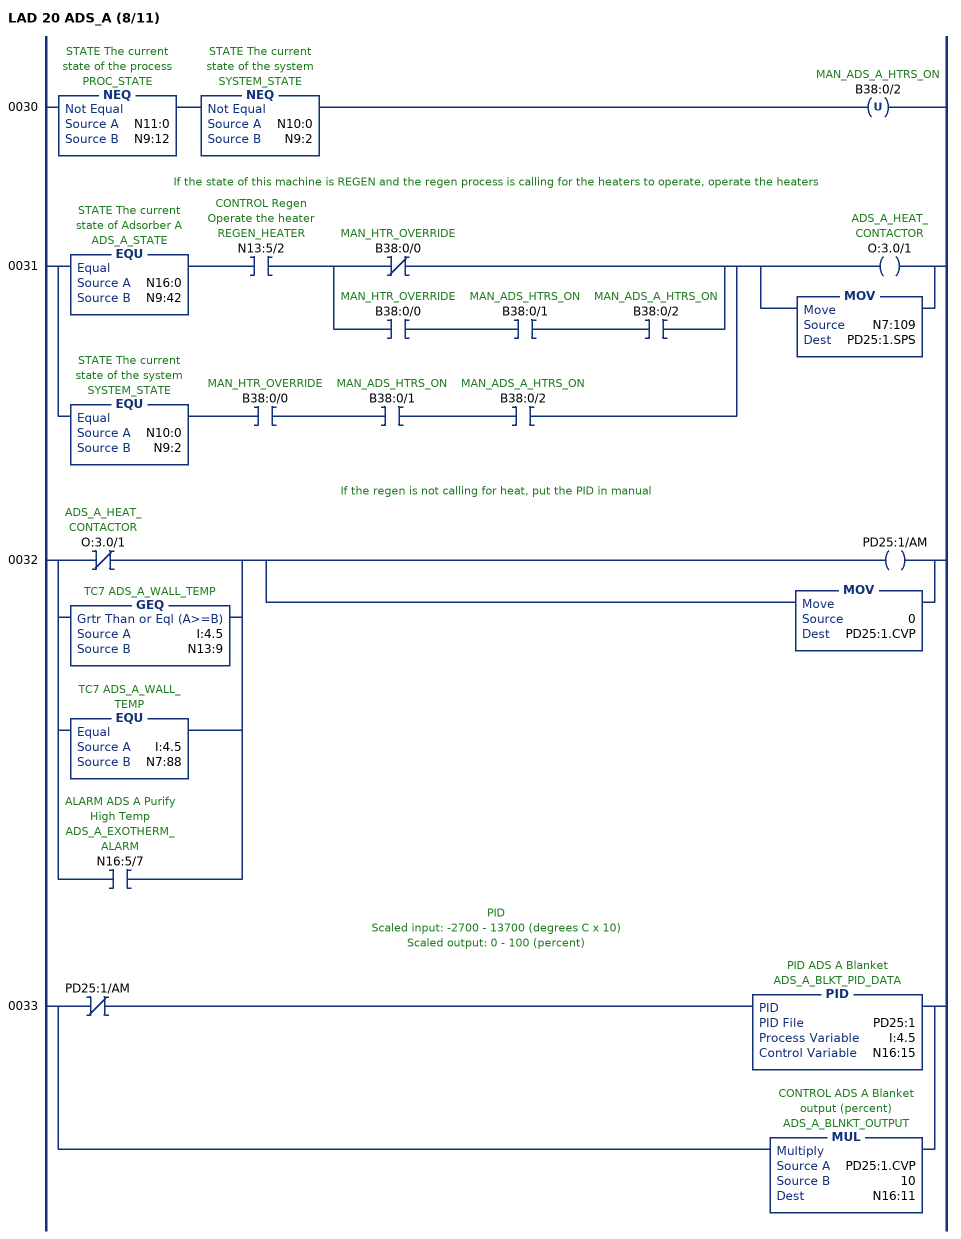
% Rung: 30 %
SOR NEQ N11:0 N9:12 NEQ N10:0 N9:2 OTU B38:0/2 EOR
%   N11:0  PROC_STATE  "STATE The current state of the process" %
%   N9:12  PROC_PURIFY_B  "STATE Process Purify B" %
%   N10:0  SYSTEM_STATE  "STATE The current state of the system" %
%   N9:2  SYSTEM_MANUAL  "STATE System Manual" %
%   B38:0/2  MAN_ADS_A_HTRS_ON %
% Rung: 31 %
% If the state of this machine is REGEN and the regen process is calling for the heaters to operate, operate the heaters %
SOR BST EQU N16:0 N9:42 XIC N13:5/2 BST XIO B38:0/0 NXB XIC B38:0/0 XIC B38:0/1 XIC B38:0/2 BND NXB EQU N10:0 N9:2 XIC B38:0/0 XIC B38:0/1 XIC B38:0/2 BND BST OTE O:3.0/1 NXB MOV N7:109 PD25:1.SPS BND EOR
%   N16:0  ADS_A_STATE  "STATE The current state of Adsorber A" %
%   N9:42  ADS_REGEN  "STATE ADS Regen" %
%   N13:5/2  REGEN_HEATER  "CONTROL Regen Operate the heater" %
%   B38:0/0  MAN_HTR_OVERRIDE %
%   B38:0/1  MAN_ADS_HTRS_ON %
%   B38:0/2  MAN_ADS_A_HTRS_ON %
%   N10:0  SYSTEM_STATE  "STATE The current state of the system" %
%   N9:2  SYSTEM_MANUAL  "STATE System Manual" %
%   O:3.0/1  ADS_A_HEAT_CONTACTOR %
%   N7:109  BLANKET_SP  "CONTROL Blanket PID Setpoint" %
% Rung: 32 %
% If the regen is not calling for heat, put the PID in manual %
SOR BST XIO O:3.0/1 NXB GEQ I:4.5 N13:9 NXB EQU I:4.5 N7:88 NXB XIC N16:5/7 BND BST OTE PD25:1/AM NXB MOV 0 PD25:1.CVP BND EOR
%   O:3.0/1  ADS_A_HEAT_CONTACTOR %
%   I:4.5  ADS_A_WALL_TEMP  "TC7" %
%   N13:9  BLANKET_LIMIT %
%   N7:88  TC_OPEN_SP  "CONFIG The value read by an open TC input" %
%   N16:5/7  ADS_A_EXOTHERM_ALARM  "ALARM ADS A Purify High Temp" %
% Rung: 33 %
% PID
% Scaled input: -2700 - 13700 (degrees C x 10)
% Scaled output: 0 - 100 (percent) %
SOR BST XIO PD25:1/AM PID PD25:1 I:4.5 N16:15 NXB MUL PD25:1.CVP 10 N16:11 BND EOR
%   PD25:1  ADS_A_BLKT_PID_DATA  "PID ADS A Blanket" %
%   I:4.5  ADS_A_WALL_TEMP  "TC7" %
%   N16:15  ADS_A_BLKT_OUTPT_RAW  "CONTROL ADS A Blanket PID Output Raw" %
%   N16:11  ADS_A_BLNKT_OUTPUT  "CONTROL ADS A Blanket output (percent)" %

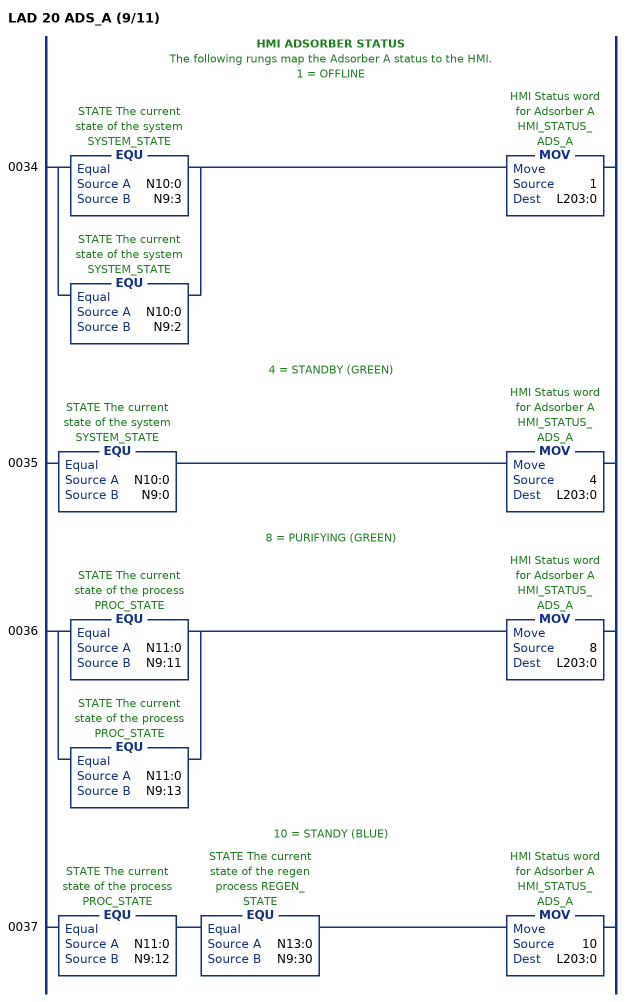
% Rung: 34 %
% TITLE: HMI ADSORBER STATUS %
% The following rungs map the Adsorber A status to the HMI.
% 1 = OFFLINE %
SOR BST EQU N10:0 N9:3 NXB EQU N10:0 N9:2 BND MOV 1 L203:0 EOR
%   N10:0  SYSTEM_STATE  "STATE The current state of the system" %
%   N9:3  SYSTEM_ALARM  "STATE System Alarm" %
%   N9:2  SYSTEM_MANUAL  "STATE System Manual" %
%   L203:0  HMI_STATUS_ADS_A  "HMI Status word for Adsorber A" %
% Rung: 35 %
% 4 = STANDBY (GREEN) %
SOR EQU N10:0 N9:0 MOV 4 L203:0 EOR
%   N10:0  SYSTEM_STATE  "STATE The current state of the system" %
%   N9:0  SYSTEM_STANDBY  "STATE System Standby" %
%   L203:0  HMI_STATUS_ADS_A  "HMI Status word for Adsorber A" %
% Rung: 36 %
% 8 = PURIFYING (GREEN) %
SOR BST EQU N11:0 N9:11 NXB EQU N11:0 N9:13 BND MOV 8 L203:0 EOR
%   N11:0  PROC_STATE  "STATE The current state of the process" %
%   N9:11  PROC_PURIFY_A  "STATE Process Purify A" %
%   N9:13  PROC_OVERLAP  "STATE Process Purify Overlap" %
%   L203:0  HMI_STATUS_ADS_A  "HMI Status word for Adsorber A" %
% Rung: 37 %
% 10 = STANDY (BLUE) %
SOR EQU N11:0 N9:12 EQU N13:0 N9:30 MOV 10 L203:0 EOR
%   N11:0  PROC_STATE  "STATE The current state of the process" %
%   N9:12  PROC_PURIFY_B  "STATE Process Purify B" %
%   N13:0  REGEN_STATE  "STATE The current state of the regen process" %
%   N9:30  REGEN_STANDBY  "STATE Regen Standby" %
%   L203:0  HMI_STATUS_ADS_A  "HMI Status word for Adsorber A" %

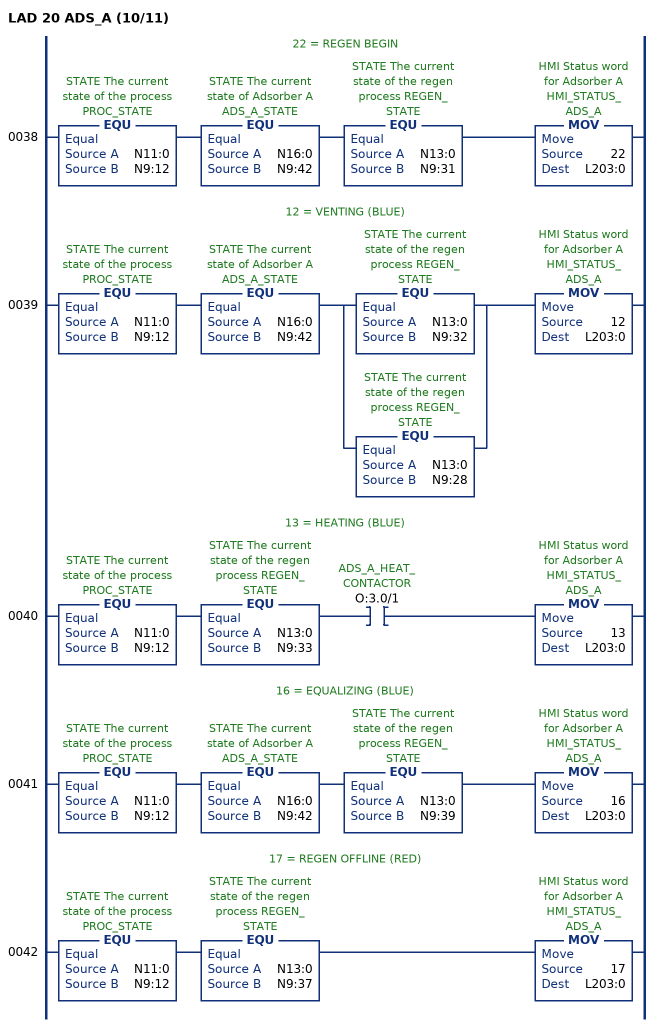
% Rung: 38 %
% 22 = REGEN BEGIN %
SOR EQU N11:0 N9:12 EQU N16:0 N9:42 EQU N13:0 N9:31 MOV 22 L203:0 EOR
%   N11:0  PROC_STATE  "STATE The current state of the process" %
%   N9:12  PROC_PURIFY_B  "STATE Process Purify B" %
%   N16:0  ADS_A_STATE  "STATE The current state of Adsorber A" %
%   N9:42  ADS_REGEN  "STATE ADS Regen" %
%   N13:0  REGEN_STATE  "STATE The current state of the regen process" %
%   N9:31  REGEN_DELAY  "STATE Regen Delay" %
%   L203:0  HMI_STATUS_ADS_A  "HMI Status word for Adsorber A" %
% Rung: 39 %
% 12 = VENTING (BLUE) %
SOR EQU N11:0 N9:12 EQU N16:0 N9:42 BST EQU N13:0 N9:32 NXB EQU N13:0 N9:28 BND MOV 12 L203:0 EOR
%   N11:0  PROC_STATE  "STATE The current state of the process" %
%   N9:12  PROC_PURIFY_B  "STATE Process Purify B" %
%   N16:0  ADS_A_STATE  "STATE The current state of Adsorber A" %
%   N9:42  ADS_REGEN  "STATE ADS Regen" %
%   N13:0  REGEN_STATE  "STATE The current state of the regen process" %
%   N9:32  REGEN_VENT  "STATE Regen Vent" %
%   N9:28  REGEN_VENT_2  "STATE Regen Vent 2" %
%   L203:0  HMI_STATUS_ADS_A  "HMI Status word for Adsorber A" %
% Rung: 40 %
% 13 = HEATING (BLUE) %
SOR EQU N11:0 N9:12 EQU N13:0 N9:33 XIC O:3.0/1 MOV 13 L203:0 EOR
%   N11:0  PROC_STATE  "STATE The current state of the process" %
%   N9:12  PROC_PURIFY_B  "STATE Process Purify B" %
%   N13:0  REGEN_STATE  "STATE The current state of the regen process" %
%   N9:33  REGEN_HEAT_BED  "STATE Regen Heat wall" %
%   O:3.0/1  ADS_A_HEAT_CONTACTOR %
%   L203:0  HMI_STATUS_ADS_A  "HMI Status word for Adsorber A" %
% Rung: 41 %
% 16 = EQUALIZING (BLUE) %
SOR EQU N11:0 N9:12 EQU N16:0 N9:42 EQU N13:0 N9:39 MOV 16 L203:0 EOR
%   N11:0  PROC_STATE  "STATE The current state of the process" %
%   N9:12  PROC_PURIFY_B  "STATE Process Purify B" %
%   N16:0  ADS_A_STATE  "STATE The current state of Adsorber A" %
%   N9:42  ADS_REGEN  "STATE ADS Regen" %
%   N13:0  REGEN_STATE  "STATE The current state of the regen process" %
%   N9:39  REGEN_EQUALIZE %
%   L203:0  HMI_STATUS_ADS_A  "HMI Status word for Adsorber A" %
% Rung: 42 %
% 17 = REGEN OFFLINE (RED) %
SOR EQU N11:0 N9:12 EQU N13:0 N9:37 MOV 17 L203:0 EOR
%   N11:0  PROC_STATE  "STATE The current state of the process" %
%   N9:12  PROC_PURIFY_B  "STATE Process Purify B" %
%   N13:0  REGEN_STATE  "STATE The current state of the regen process" %
%   N9:37  REGEN_ALARM  "STATE Regen Alarm" %
%   L203:0  HMI_STATUS_ADS_A  "HMI Status word for Adsorber A" %

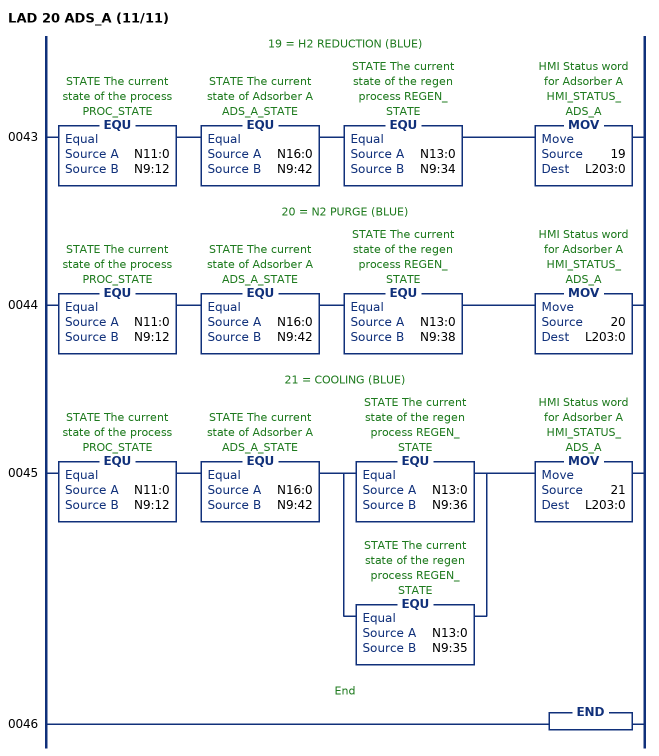
% Rung: 43 %
% 19 = H2 REDUCTION (BLUE) %
SOR EQU N11:0 N9:12 EQU N16:0 N9:42 EQU N13:0 N9:34 MOV 19 L203:0 EOR
%   N11:0  PROC_STATE  "STATE The current state of the process" %
%   N9:12  PROC_PURIFY_B  "STATE Process Purify B" %
%   N16:0  ADS_A_STATE  "STATE The current state of Adsorber A" %
%   N9:42  ADS_REGEN  "STATE ADS Regen" %
%   N13:0  REGEN_STATE  "STATE The current state of the regen process" %
%   N9:34  REGEN_H2_REDUCTION  "STATE Regen Running" %
%   L203:0  HMI_STATUS_ADS_A  "HMI Status word for Adsorber A" %
% Rung: 44 %
% 20 = N2 PURGE (BLUE) %
SOR EQU N11:0 N9:12 EQU N16:0 N9:42 EQU N13:0 N9:38 MOV 20 L203:0 EOR
%   N11:0  PROC_STATE  "STATE The current state of the process" %
%   N9:12  PROC_PURIFY_B  "STATE Process Purify B" %
%   N16:0  ADS_A_STATE  "STATE The current state of Adsorber A" %
%   N9:42  ADS_REGEN  "STATE ADS Regen" %
%   N13:0  REGEN_STATE  "STATE The current state of the regen process" %
%   N9:38  REGEN_PURGE  "STATE Regen Hot Purge" %
%   L203:0  HMI_STATUS_ADS_A  "HMI Status word for Adsorber A" %
% Rung: 45 %
% 21 = COOLING (BLUE) %
SOR EQU N11:0 N9:12 EQU N16:0 N9:42 BST EQU N13:0 N9:36 NXB EQU N13:0 N9:35 BND MOV 21 L203:0 EOR
%   N11:0  PROC_STATE  "STATE The current state of the process" %
%   N9:12  PROC_PURIFY_B  "STATE Process Purify B" %
%   N16:0  ADS_A_STATE  "STATE The current state of Adsorber A" %
%   N9:42  ADS_REGEN  "STATE ADS Regen" %
%   N13:0  REGEN_STATE  "STATE The current state of the regen process" %
%   N9:36  REGEN_COOL  "STATE Regen Cool" %
%   N9:35  REGEN_COOL_WALL  "STATE Regen Cool wall" %
%   L203:0  HMI_STATUS_ADS_A  "HMI Status word for Adsorber A" %
% Rung: 46 %
% End %
SOR END EOR

LADDER 21 "ADS_A_FLT"    % Controls the Adsorber A faults %
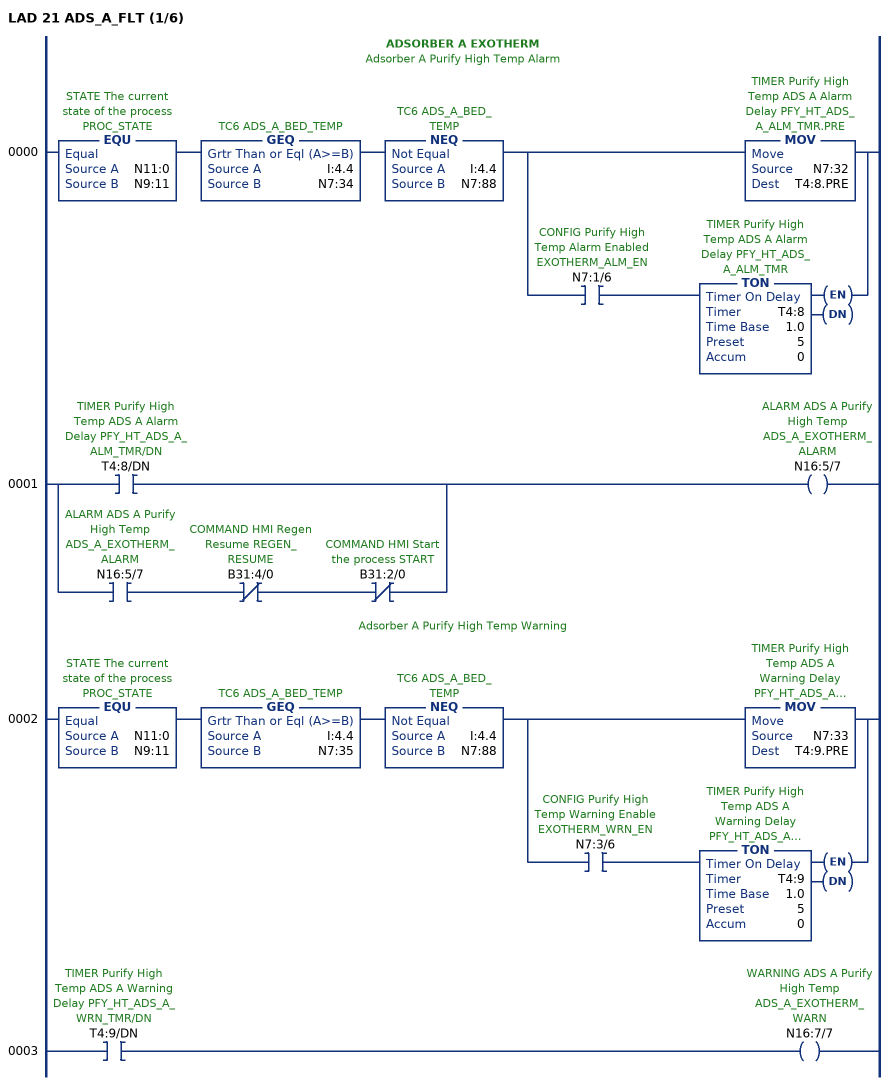
% Rung: 0 %
% TITLE: ADSORBER A EXOTHERM %
% Adsorber A Purify High Temp Alarm %
SOR EQU N11:0 N9:11 GEQ I:4.4 N7:34 NEQ I:4.4 N7:88 BST MOV N7:32 T4:8.PRE NXB XIC N7:1/6 TON T4:8 1.0 5 0 BND EOR
%   N11:0  PROC_STATE  "STATE The current state of the process" %
%   N9:11  PROC_PURIFY_A  "STATE Process Purify A" %
%   I:4.4  ADS_A_BED_TEMP  "TC6" %
%   N7:34  EXOTHERM_ALM_SP  "CONFIG Purify High Temp Alarm Setpoint" %
%   N7:88  TC_OPEN_SP  "CONFIG The value read by an open TC input" %
%   N7:32  EXOTHERM_ALM_DLY  "CONFIG Purify High Temp Alarm Delay" %
%   T4:8  PFY_HT_ADS_A_ALM_TMR  "TIMER Purify High Temp ADS A Alarm Delay" %
%   N7:1/6  EXOTHERM_ALM_EN  "CONFIG Purify High Temp Alarm Enabled" %
% Rung: 1 %
SOR BST XIC T4:8/DN NXB XIC N16:5/7 XIO B31:4/0 XIO B31:2/0 BND OTE N16:5/7 EOR
%   T4:8  PFY_HT_ADS_A_ALM_TMR  "TIMER Purify High Temp ADS A Alarm Delay" %
%   N16:5/7  ADS_A_EXOTHERM_ALARM  "ALARM ADS A Purify High Temp" %
%   B31:4/0  REGEN_RESUME  "COMMAND HMI Regen Resume" %
%   B31:2/0  START  "COMMAND HMI Start the process" %
% Rung: 2 %
% Adsorber A Purify High Temp Warning %
SOR EQU N11:0 N9:11 GEQ I:4.4 N7:35 NEQ I:4.4 N7:88 BST MOV N7:33 T4:9.PRE NXB XIC N7:3/6 TON T4:9 1.0 5 0 BND EOR
%   N11:0  PROC_STATE  "STATE The current state of the process" %
%   N9:11  PROC_PURIFY_A  "STATE Process Purify A" %
%   I:4.4  ADS_A_BED_TEMP  "TC6" %
%   N7:35  EXOTHERM_WRN_SP  "CONFIG Purify High Temp Warning Setpoint" %
%   N7:88  TC_OPEN_SP  "CONFIG The value read by an open TC input" %
%   N7:33  EXOTHERM_WRN_DLY  "CONFIG Purify High Temp Warning Delay" %
%   T4:9  PFY_HT_ADS_A_WRN_TMR  "TIMER Purify High Temp ADS A Warning Delay" %
%   N7:3/6  EXOTHERM_WRN_EN  "CONFIG Purify High Temp Warning Enable" %
% Rung: 3 %
SOR XIC T4:9/DN OTE N16:7/7 EOR
%   T4:9  PFY_HT_ADS_A_WRN_TMR  "TIMER Purify High Temp ADS A Warning Delay" %
%   N16:7/7  ADS_A_EXOTHERM_WARN  "WARNING ADS A Purify High Temp" %

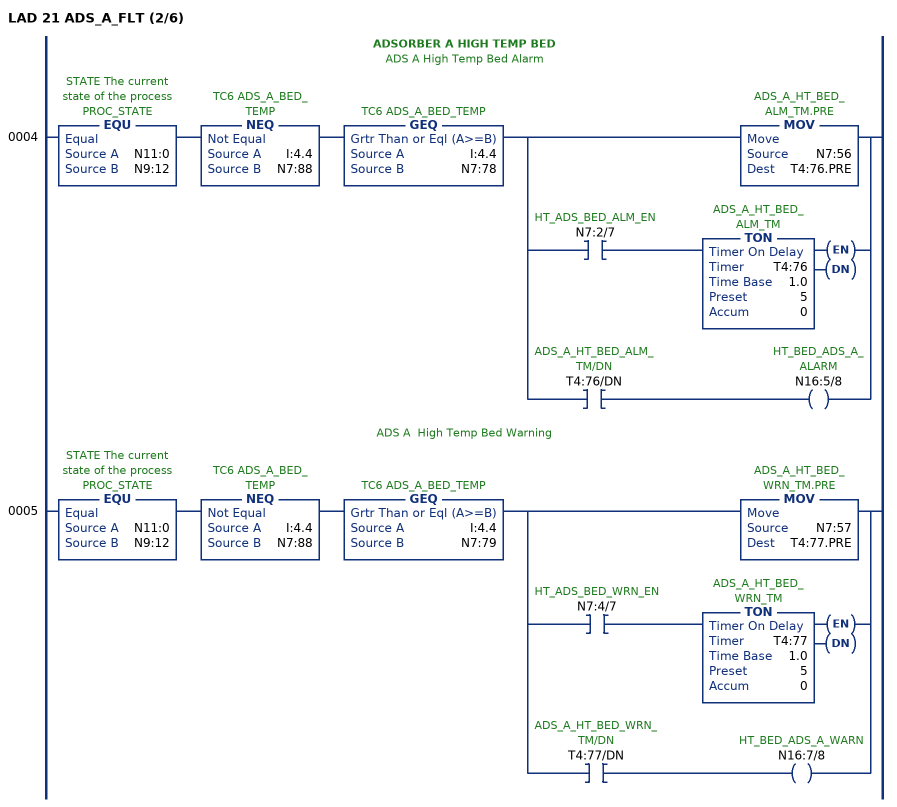
% Rung: 4 %
% TITLE: ADSORBER A HIGH TEMP BED %
% ADS A High Temp Bed Alarm %
SOR EQU N11:0 N9:12 NEQ I:4.4 N7:88 GEQ I:4.4 N7:78 BST MOV N7:56 T4:76.PRE NXB XIC N7:2/7 TON T4:76 1.0 5 0 NXB XIC T4:76/DN OTE N16:5/8 BND EOR
%   N11:0  PROC_STATE  "STATE The current state of the process" %
%   N9:12  PROC_PURIFY_B  "STATE Process Purify B" %
%   I:4.4  ADS_A_BED_TEMP  "TC6" %
%   N7:88  TC_OPEN_SP  "CONFIG The value read by an open TC input" %
%   N7:78  HT_ADS_BED_ALM_SP %
%   N7:56  HT_ADS_BED_ALM_DLY %
%   T4:76  ADS_A_HT_BED_ALM_TM %
%   N7:2/7  HT_ADS_BED_ALM_EN %
%   N16:5/8  HT_BED_ADS_A_ALARM %
% Rung: 5 %
% ADS A  High Temp Bed Warning %
SOR EQU N11:0 N9:12 NEQ I:4.4 N7:88 GEQ I:4.4 N7:79 BST MOV N7:57 T4:77.PRE NXB XIC N7:4/7 TON T4:77 1.0 5 0 NXB XIC T4:77/DN OTE N16:7/8 BND EOR
%   N11:0  PROC_STATE  "STATE The current state of the process" %
%   N9:12  PROC_PURIFY_B  "STATE Process Purify B" %
%   I:4.4  ADS_A_BED_TEMP  "TC6" %
%   N7:88  TC_OPEN_SP  "CONFIG The value read by an open TC input" %
%   N7:79  HT_ADS_BED_WRN_SP %
%   N7:57  HT_ADS_BED_WRN_DLY %
%   T4:77  ADS_A_HT_BED_WRN_TM %
%   N7:4/7  HT_ADS_BED_WRN_EN %
%   N16:7/8  HT_BED_ADS_A_WARN %

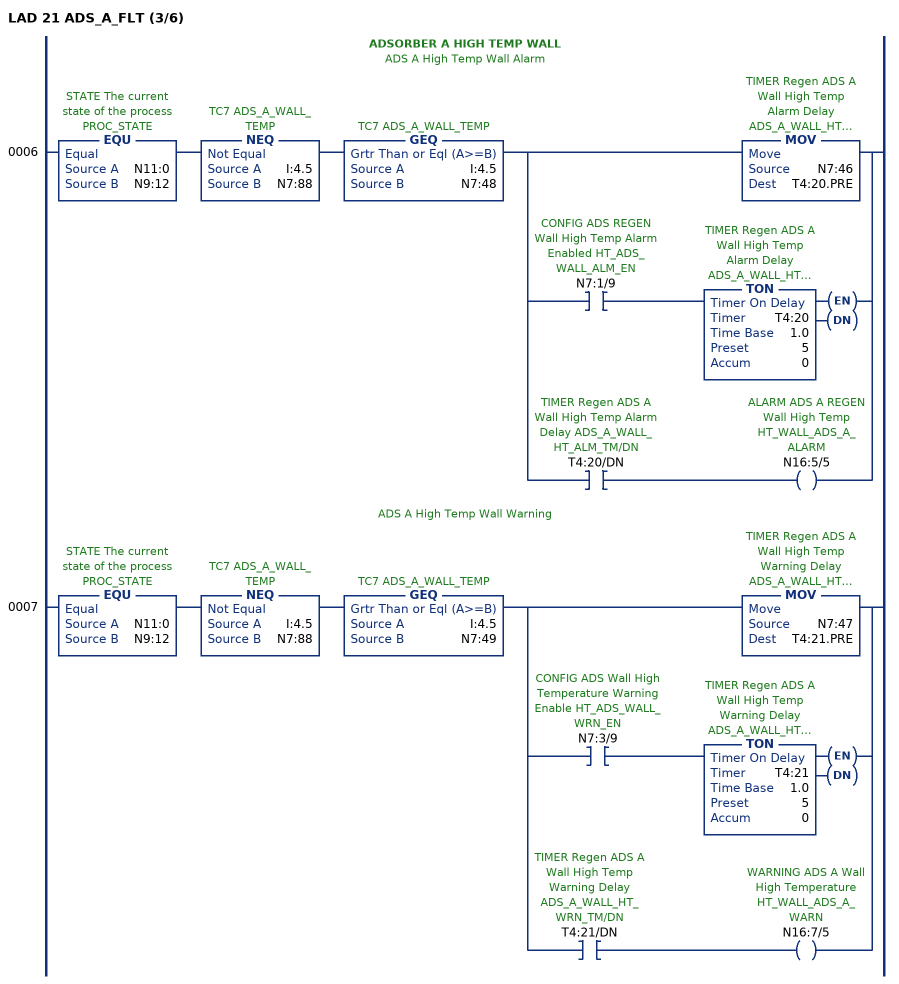
% Rung: 6 %
% TITLE: ADSORBER A HIGH TEMP WALL %
% ADS A High Temp Wall Alarm %
SOR EQU N11:0 N9:12 NEQ I:4.5 N7:88 GEQ I:4.5 N7:48 BST MOV N7:46 T4:20.PRE NXB XIC N7:1/9 TON T4:20 1.0 5 0 NXB XIC T4:20/DN OTE N16:5/5 BND EOR
%   N11:0  PROC_STATE  "STATE The current state of the process" %
%   N9:12  PROC_PURIFY_B  "STATE Process Purify B" %
%   I:4.5  ADS_A_WALL_TEMP  "TC7" %
%   N7:88  TC_OPEN_SP  "CONFIG The value read by an open TC input" %
%   N7:48  HT_ADS_WALL_ALM_SP  "CONFIG ADS Wall Regen High Temp Alarm" %
%   N7:46  HT_ADS_WALL_ALM_DLY  "CONFIG ADS Wall High Temperature Alarm Delay" %
%   T4:20  ADS_A_WALL_HT_ALM_TM  "TIMER Regen ADS A Wall High Temp Alarm Delay" %
%   N7:1/9  HT_ADS_WALL_ALM_EN  "CONFIG ADS REGEN Wall High Temp Alarm Enabled" %
%   N16:5/5  HT_WALL_ADS_A_ALARM  "ALARM ADS A REGEN Wall High Temp" %
% Rung: 7 %
% ADS A High Temp Wall Warning %
SOR EQU N11:0 N9:12 NEQ I:4.5 N7:88 GEQ I:4.5 N7:49 BST MOV N7:47 T4:21.PRE NXB XIC N7:3/9 TON T4:21 1.0 5 0 NXB XIC T4:21/DN OTE N16:7/5 BND EOR
%   N11:0  PROC_STATE  "STATE The current state of the process" %
%   N9:12  PROC_PURIFY_B  "STATE Process Purify B" %
%   I:4.5  ADS_A_WALL_TEMP  "TC7" %
%   N7:88  TC_OPEN_SP  "CONFIG The value read by an open TC input" %
%   N7:49  HT_ADS_WALL_WRN_SP  "CONFIG ADS Wall Regen High Temp Alarm" %
%   N7:47  HT_ADS_WALL_WRN_DLY  "CONFIG ADS Wall High Temperature Warning Delay" %
%   T4:21  ADS_A_WALL_HT_WRN_TM  "TIMER Regen ADS A Wall High Temp Warning Delay" %
%   N7:3/9  HT_ADS_WALL_WRN_EN  "CONFIG ADS Wall High Temperature Warning Enable" %
%   N16:7/5  HT_WALL_ADS_A_WARN  "WARNING ADS A Wall High Temperature" %

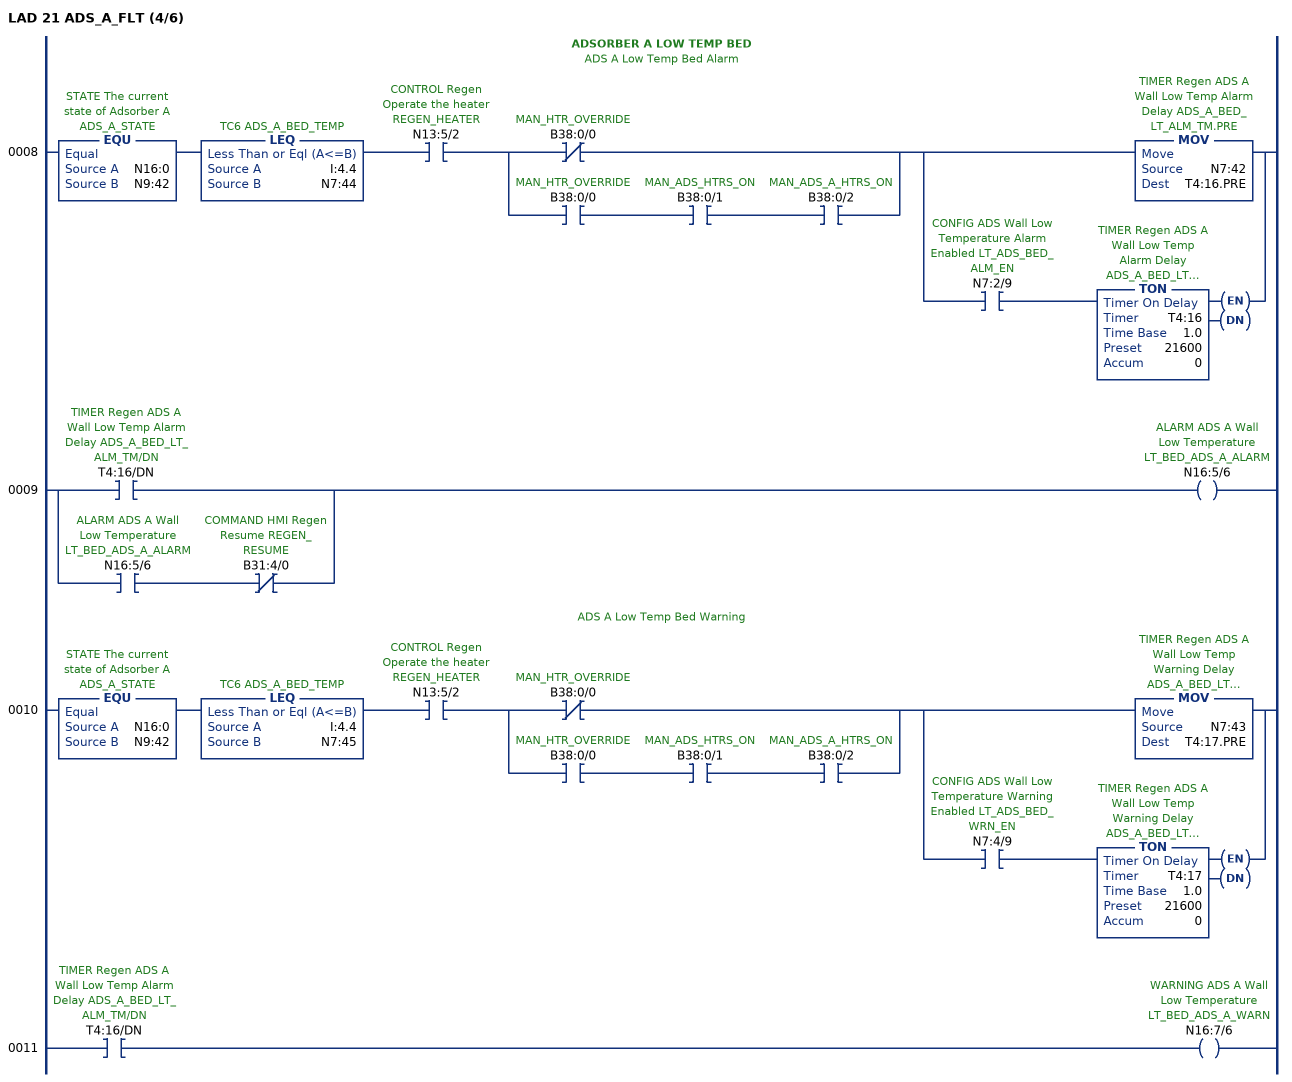
% Rung: 8 %
% TITLE: ADSORBER A LOW TEMP BED %
% ADS A Low Temp Bed Alarm %
SOR EQU N16:0 N9:42 LEQ I:4.4 N7:44 XIC N13:5/2 BST XIO B38:0/0 NXB XIC B38:0/0 XIC B38:0/1 XIC B38:0/2 BND BST MOV N7:42 T4:16.PRE NXB XIC N7:2/9 TON T4:16 1.0 21600 0 BND EOR
%   N16:0  ADS_A_STATE  "STATE The current state of Adsorber A" %
%   N9:42  ADS_REGEN  "STATE ADS Regen" %
%   I:4.4  ADS_A_BED_TEMP  "TC6" %
%   N7:44  LT_ADS_BED_ALM_SP  "CONFIG ADS Wall Regen Heat Low Temperature Alarm Setpoint" %
%   N13:5/2  REGEN_HEATER  "CONTROL Regen Operate the heater" %
%   B38:0/0  MAN_HTR_OVERRIDE %
%   B38:0/1  MAN_ADS_HTRS_ON %
%   B38:0/2  MAN_ADS_A_HTRS_ON %
%   N7:42  LT_ADS_BED_ALM_DLY  "CONFIG ADS Wall Regen heat Low Temperature Alarm Delay" %
%   T4:16  ADS_A_BED_LT_ALM_TM  "TIMER Regen ADS A Wall Low Temp Alarm Delay" %
%   N7:2/9  LT_ADS_BED_ALM_EN  "CONFIG ADS Wall Low Temperature Alarm Enabled" %
% Rung: 9 %
SOR BST XIC T4:16/DN NXB XIC N16:5/6 XIO B31:4/0 BND OTE N16:5/6 EOR
%   T4:16  ADS_A_BED_LT_ALM_TM  "TIMER Regen ADS A Wall Low Temp Alarm Delay" %
%   N16:5/6  LT_BED_ADS_A_ALARM  "ALARM ADS A Wall Low Temperature" %
%   B31:4/0  REGEN_RESUME  "COMMAND HMI Regen Resume" %
% Rung: 10 %
% ADS A Low Temp Bed Warning %
SOR EQU N16:0 N9:42 LEQ I:4.4 N7:45 XIC N13:5/2 BST XIO B38:0/0 NXB XIC B38:0/0 XIC B38:0/1 XIC B38:0/2 BND BST MOV N7:43 T4:17.PRE NXB XIC N7:4/9 TON T4:17 1.0 21600 0 BND EOR
%   N16:0  ADS_A_STATE  "STATE The current state of Adsorber A" %
%   N9:42  ADS_REGEN  "STATE ADS Regen" %
%   I:4.4  ADS_A_BED_TEMP  "TC6" %
%   N7:45  LT_ADS_BED_WRN_SP  "CONFIG ADS Wall Regen Heat Low Temperature Warning Setpoint" %
%   N13:5/2  REGEN_HEATER  "CONTROL Regen Operate the heater" %
%   B38:0/0  MAN_HTR_OVERRIDE %
%   B38:0/1  MAN_ADS_HTRS_ON %
%   B38:0/2  MAN_ADS_A_HTRS_ON %
%   N7:43  LT_ADS_BED_WRN_DLY  "CONFIG ADS Wall Regen heat Low Temperature Warning Delay" %
%   T4:17  ADS_A_BED_LT_WRN_TM  "TIMER Regen ADS A Wall Low Temp Warning Delay" %
%   N7:4/9  LT_ADS_BED_WRN_EN  "CONFIG ADS Wall Low Temperature Warning Enabled" %
% Rung: 11 %
SOR XIC T4:16/DN OTE N16:7/6 EOR
%   T4:16  ADS_A_BED_LT_ALM_TM  "TIMER Regen ADS A Wall Low Temp Alarm Delay" %
%   N16:7/6  LT_BED_ADS_A_WARN  "WARNING ADS A Wall Low Temperature" %

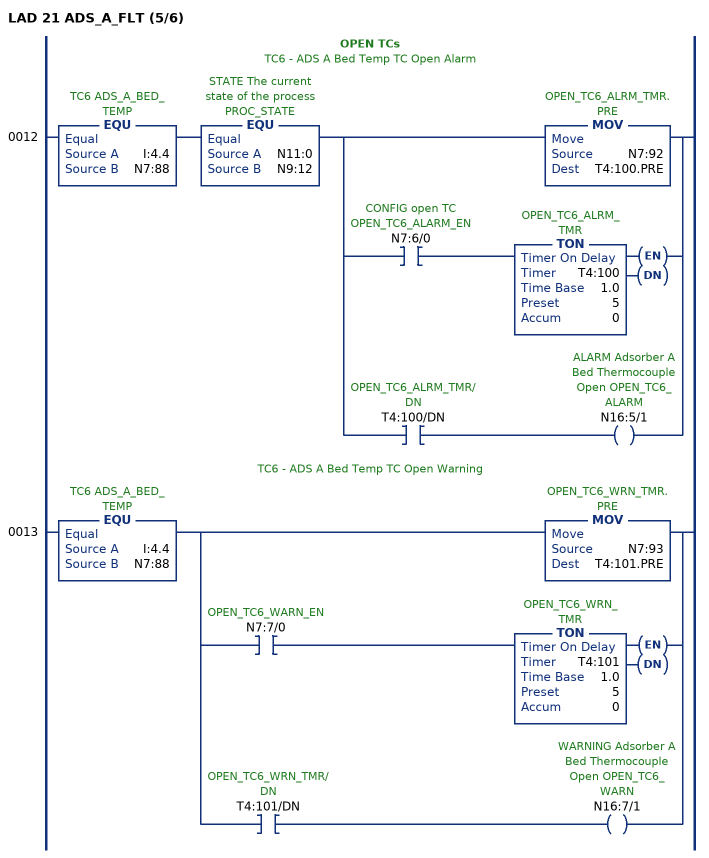
% Rung: 12 %
% TITLE: OPEN TCs %
% TC6 - ADS A Bed Temp TC Open Alarm %
SOR EQU I:4.4 N7:88 EQU N11:0 N9:12 BST MOV N7:92 T4:100.PRE NXB BST XIC N7:6/0 TON T4:100 1.0 5 0 NXB XIC T4:100/DN OTE N16:5/1 BND BND EOR
%   I:4.4  ADS_A_BED_TEMP  "TC6" %
%   N7:88  TC_OPEN_SP  "CONFIG The value read by an open TC input" %
%   N11:0  PROC_STATE  "STATE The current state of the process" %
%   N9:12  PROC_PURIFY_B  "STATE Process Purify B" %
%   N7:92  OPEN_TC_ALARM_DELAY %
%   T4:100  OPEN_TC6_ALRM_TMR %
%   N7:6/0  OPEN_TC6_ALARM_EN  "CONFIG open TC" %
%   N16:5/1  OPEN_TC6_ALARM  "ALARM Adsorber A Bed Thermocouple Open" %
% Rung: 13 %
% TC6 - ADS A Bed Temp TC Open Warning %
SOR EQU I:4.4 N7:88 BST MOV N7:93 T4:101.PRE NXB BST XIC N7:7/0 TON T4:101 1.0 5 0 NXB XIC T4:101/DN OTE N16:7/1 BND BND EOR
%   I:4.4  ADS_A_BED_TEMP  "TC6" %
%   N7:88  TC_OPEN_SP  "CONFIG The value read by an open TC input" %
%   N7:93  OPEN_TC_WRN_DELAY %
%   T4:101  OPEN_TC6_WRN_TMR %
%   N7:7/0  OPEN_TC6_WARN_EN %
%   N16:7/1  OPEN_TC6_WARN  "WARNING Adsorber A Bed Thermocouple Open" %

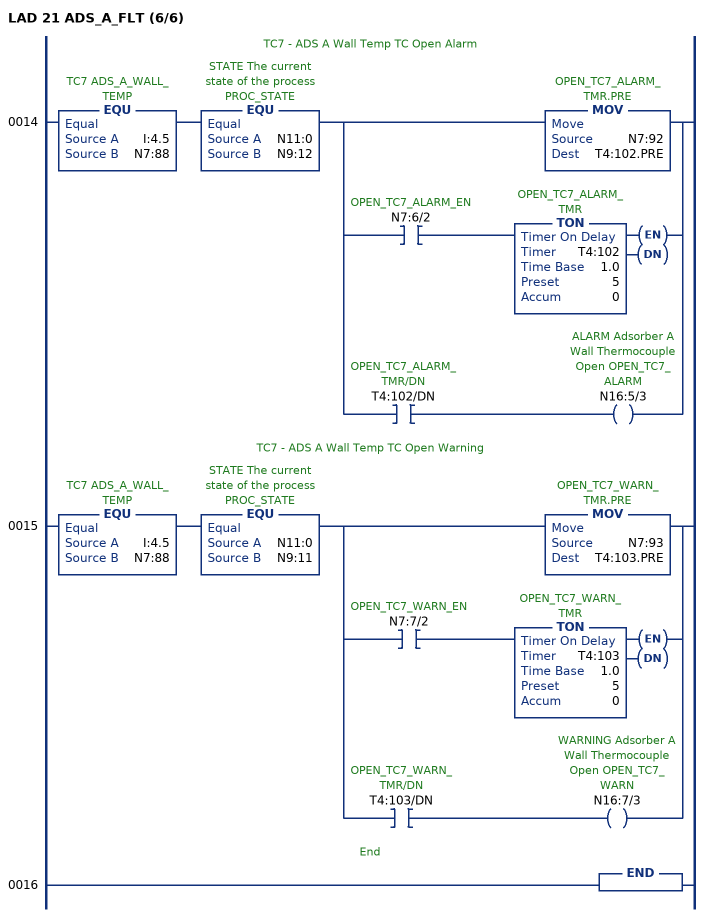
% Rung: 14 %
% TC7 - ADS A Wall Temp TC Open Alarm %
SOR EQU I:4.5 N7:88 EQU N11:0 N9:12 BST MOV N7:92 T4:102.PRE NXB BST XIC N7:6/2 TON T4:102 1.0 5 0 NXB XIC T4:102/DN OTE N16:5/3 BND BND EOR
%   I:4.5  ADS_A_WALL_TEMP  "TC7" %
%   N7:88  TC_OPEN_SP  "CONFIG The value read by an open TC input" %
%   N11:0  PROC_STATE  "STATE The current state of the process" %
%   N9:12  PROC_PURIFY_B  "STATE Process Purify B" %
%   N7:92  OPEN_TC_ALARM_DELAY %
%   T4:102  OPEN_TC7_ALARM_TMR %
%   N7:6/2  OPEN_TC7_ALARM_EN %
%   N16:5/3  OPEN_TC7_ALARM  "ALARM Adsorber A Wall Thermocouple Open" %
% Rung: 15 %
% TC7 - ADS A Wall Temp TC Open Warning %
SOR EQU I:4.5 N7:88 EQU N11:0 N9:11 BST MOV N7:93 T4:103.PRE NXB BST XIC N7:7/2 TON T4:103 1.0 5 0 NXB XIC T4:103/DN OTE N16:7/3 BND BND EOR
%   I:4.5  ADS_A_WALL_TEMP  "TC7" %
%   N7:88  TC_OPEN_SP  "CONFIG The value read by an open TC input" %
%   N11:0  PROC_STATE  "STATE The current state of the process" %
%   N9:11  PROC_PURIFY_A  "STATE Process Purify A" %
%   N7:93  OPEN_TC_WRN_DELAY %
%   T4:103  OPEN_TC7_WARN_TMR %
%   N7:7/2  OPEN_TC7_WARN_EN %
%   N16:7/3  OPEN_TC7_WARN  "WARNING Adsorber A Wall Thermocouple Open" %
% Rung: 16 %
% End %
SOR END EOR

LADDER 22 "ADS_B"    % Controld Adsorber B %
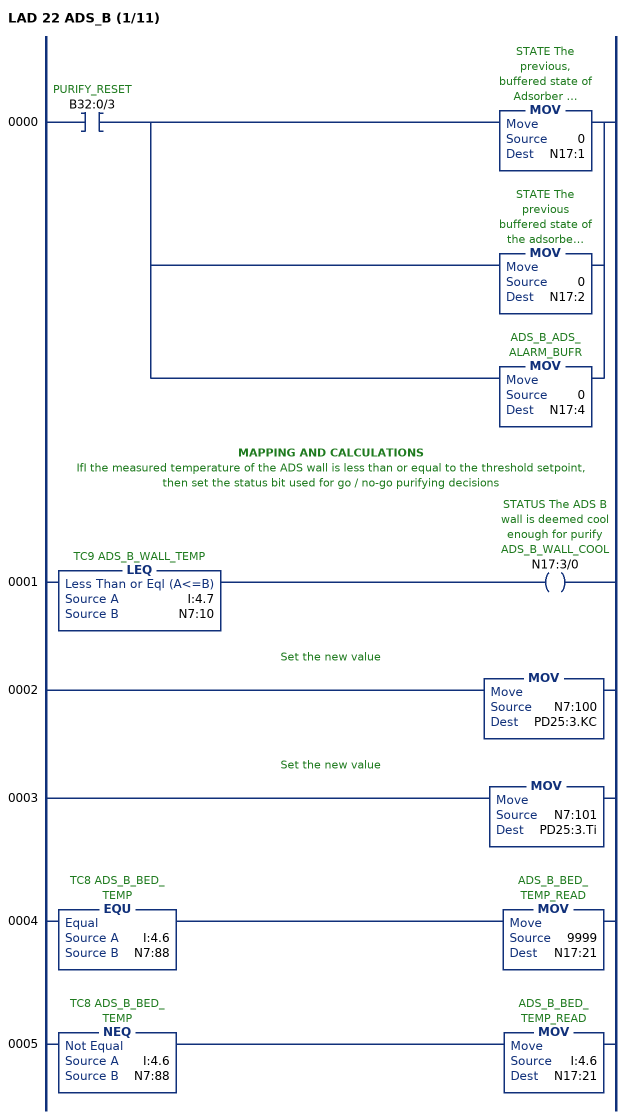
% Rung: 0 %
SOR XIC B32:0/3 BST MOV 0 N17:1 NXB MOV 0 N17:2 NXB MOV 0 N17:4 BND EOR
%   B32:0/3  PURIFY_RESET %
%   N17:1  ADS_B_STANDBY_BUFFER  "STATE The previous, buffered state of Adsorber B" %
%   N17:2  ADS_B_SYS_ALARM_BUFR  "STATE The previous buffered state of the adsorber when the alarm occured" %
%   N17:4  ADS_B_ADS_ALARM_BUFR %
% Rung: 1 %
% TITLE: MAPPING AND CALCULATIONS %
% IfI the measured temperature of the ADS wall is less than or equal to the threshold setpoint, then set the status bit used for go / no-go purifying decisions %
SOR LEQ I:4.7 N7:10 OTE N17:3/0 EOR
%   I:4.7  ADS_B_WALL_TEMP  "TC9" %
%   N7:10  ADS_WALL_TEMP_COOL  "CONFIG The temp at which the adsorber wall is deemed to be cool enough to purify" %
%   N17:3/0  ADS_B_WALL_COOL  "STATUS The ADS B wall is deemed cool enough for purify" %
% Rung: 2 %
% Set the new value %
SOR MOV N7:100 PD25:3.KC EOR
%   N7:100  BLANKET_P  "CONFIG Blanket Proportional Gain New" %
% Rung: 3 %
% Set the new value %
SOR MOV N7:101 PD25:3.Ti EOR
%   N7:101  BLANKET_I  "CONFIG Blanket Integral Gain New" %
% Rung: 4 %
SOR EQU I:4.6 N7:88 MOV 9999 N17:21 EOR
%   I:4.6  ADS_B_BED_TEMP  "TC8" %
%   N7:88  TC_OPEN_SP  "CONFIG The value read by an open TC input" %
%   N17:21  ADS_B_BED_TEMP_READ %
% Rung: 5 %
SOR NEQ I:4.6 N7:88 MOV I:4.6 N17:21 EOR
%   I:4.6  ADS_B_BED_TEMP  "TC8" %
%   N7:88  TC_OPEN_SP  "CONFIG The value read by an open TC input" %
%   N17:21  ADS_B_BED_TEMP_READ %

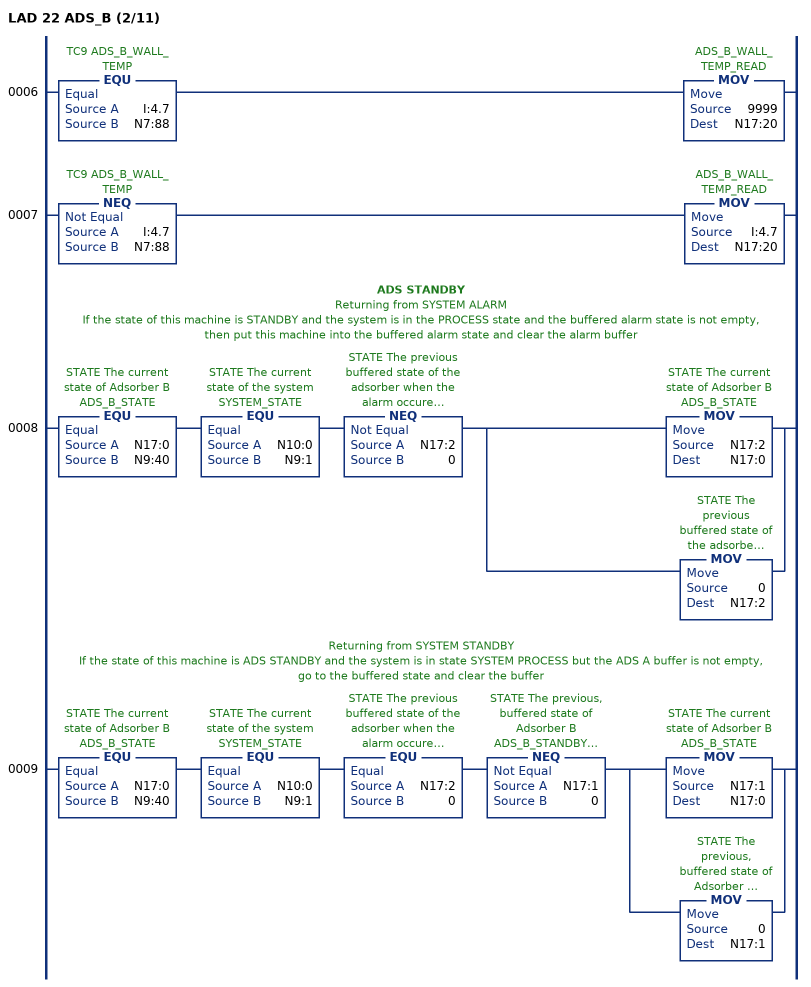
% Rung: 6 %
SOR EQU I:4.7 N7:88 MOV 9999 N17:20 EOR
%   I:4.7  ADS_B_WALL_TEMP  "TC9" %
%   N7:88  TC_OPEN_SP  "CONFIG The value read by an open TC input" %
%   N17:20  ADS_B_WALL_TEMP_READ %
% Rung: 7 %
SOR NEQ I:4.7 N7:88 MOV I:4.7 N17:20 EOR
%   I:4.7  ADS_B_WALL_TEMP  "TC9" %
%   N7:88  TC_OPEN_SP  "CONFIG The value read by an open TC input" %
%   N17:20  ADS_B_WALL_TEMP_READ %
% Rung: 8 %
% TITLE: ADS STANDBY %
% Returning from SYSTEM ALARM
% If the state of this machine is STANDBY and the system is in the PROCESS state and the buffered alarm state is not empty, then put this machine into the buffered alarm state and clear the alarm buffer %
SOR EQU N17:0 N9:40 EQU N10:0 N9:1 NEQ N17:2 0 BST MOV N17:2 N17:0 NXB MOV 0 N17:2 BND EOR
%   N17:0  ADS_B_STATE  "STATE The current state of Adsorber B" %
%   N9:40  ADS_STANDBY  "STATE ADS Standby" %
%   N10:0  SYSTEM_STATE  "STATE The current state of the system" %
%   N9:1  SYSTEM_PROCESS  "STATE System Process" %
%   N17:2  ADS_B_SYS_ALARM_BUFR  "STATE The previous buffered state of the adsorber when the alarm occured" %
% Rung: 9 %
% Returning from SYSTEM STANDBY
% If the state of this machine is ADS STANDBY and the system is in state SYSTEM PROCESS but the ADS A buffer is not empty, go to the buffered state and clear the buffer %
SOR EQU N17:0 N9:40 EQU N10:0 N9:1 EQU N17:2 0 NEQ N17:1 0 BST MOV N17:1 N17:0 NXB MOV 0 N17:1 BND EOR
%   N17:0  ADS_B_STATE  "STATE The current state of Adsorber B" %
%   N9:40  ADS_STANDBY  "STATE ADS Standby" %
%   N10:0  SYSTEM_STATE  "STATE The current state of the system" %
%   N9:1  SYSTEM_PROCESS  "STATE System Process" %
%   N17:2  ADS_B_SYS_ALARM_BUFR  "STATE The previous buffered state of the adsorber when the alarm occured" %
%   N17:1  ADS_B_STANDBY_BUFFER  "STATE The previous, buffered state of Adsorber B" %

